// TIA Portal project "HW_2000528_main_V18" (V18)

(* hardware
DEVICE "GSD device_4"  GSD.Device.PN
   slot 0: "Rack"  Rack  V1.0
   slot 0: "CPX_WP5_L"  CPX Rev 30  TN 197330  V4.2.30
      slot 0: "CPX Rev 30"  CPX Rev 30
      slot 1: "PN-IO Interface"  PN-IO Interface
         slot 1: "Port 1"  Port 1
         slot 2: "Port 2"  Port 2
   slot 1: "FB33 PNIO Module_1"  FB33 PNIO Module  TN 548755, CPX-FB33, Code F33
      slot 0: "FB33 PNIO Module"  FB33 PNIO Module
   slot 2: "MPA1S VMPA1-FB-EMS-8 [8DO]_1"  MPA1S VMPA1-FB-EMS-8 [8DO]  TN 533360, VMPA1-FB-EMS-8, Code A
      slot 0: "MPA1S VMPA1-FB-EMS-8 [8DO]"  MPA1S VMPA1-FB-EMS-8 [8DO]
   slot 3: "MPA1S VMPA1-FB-EMS-8 [8DO]_2"  MPA1S VMPA1-FB-EMS-8 [8DO]  TN 533360, VMPA1-FB-EMS-8, Code A
      slot 0: "MPA1S VMPA1-FB-EMS-8 [8DO]"  MPA1S VMPA1-FB-EMS-8 [8DO]
   slot 4: "MPA1S VMPA1-FB-EMS-8 [8DO]_3"  MPA1S VMPA1-FB-EMS-8 [8DO]  TN 533360, VMPA1-FB-EMS-8, Code A
      slot 0: "MPA1S VMPA1-FB-EMS-8 [8DO]"  MPA1S VMPA1-FB-EMS-8 [8DO]
DEVICE "GSD device_2"  GSD.Device.PN
   slot 0: "WP002-DM260-L"  DataMan 260  DMR-260#-#0  5.5.0
      slot 0: "DataMan 260"  DataMan 260
      slot 1: "Interface"  Interface
         slot 1: "Port 1"  Port 1
   slot 0: "Rack"  Rack  V1.0
   slot 1: "Acquisition Control_1"  Acquisition Control
      slot 0: "Acquisition Control"  Acquisition Control
   slot 2: "Acquisition Status_1"  Acquisition Status
      slot 0: "Acquisition Status"  Acquisition Status
   slot 3: "Results Control_1"  Results Control
      slot 0: "Results Control"  Results Control
   slot 4: "Results Status_1"  Results Status
      slot 0: "Results Status"  Results Status
   slot 5: "Soft Event Control_1"  Soft Event Control
      slot 0: "Soft Event Control"  Soft Event Control
   slot 6: "User Data - 64 bytes_1"  User Data - 64 bytes
      slot 0: "User Data - 64 bytes"  User Data - 64 bytes
   slot 7: "Result Data - 64 bytes_1"  Result Data - 64 bytes
      slot 0: "Result Data - 64 bytes"  Result Data - 64 bytes
DEVICE "ET 200SP station_5"  ET 200SP-Station
   slot 0: "R6_L"  IM 155-6 PN ST  6ES7 155-6AU01-0BN0  V4.1
   slot 0: "Rack_0"  Rack  6ES5 710-8MAx1
   slot 1: "DI 16x24VDC ST_1"  DI 16x24VDC ST  6ES7 131-6BH01-0BA0  V0.0
      slot 1: "DI 16x24VDC ST_1"  DI 16x24VDC ST
   slot 2: "DI 16x24VDC ST_2"  DI 16x24VDC ST  6ES7 131-6BH01-0BA0  V0.0
      slot 1: "DI 16x24VDC ST_2"  DI 16x24VDC ST
   slot 3: "DQ 16x24VDC/0.5A ST_1"  DQ 16x24VDC/0.5A ST  6ES7 132-6BH01-0BA0  V0.0
      slot 1: "DQ 16x24VDC/0.5A ST_1"  DQ 16x24VDC/0.5A ST
   slot 4: "DQ 16x24VDC/0.5A ST_2"  DQ 16x24VDC/0.5A ST  6ES7 132-6BH01-0BA0  V0.0
      slot 1: "DQ 16x24VDC/0.5A ST_2"  DQ 16x24VDC/0.5A ST
   slot 5: "Server module_1"  Server module  6ES7 193-6PA00-0AA0  V1.1
      slot 1: "Server module_1"  Server module
   slot 127: "BA 2xRJ45"  BA 2xRJ45  6ES7 193-6AR00-0AA0  V0.0
      slot 1: "Port_1"  X1 P1 R  6ES7 193-6AR00-0AA0  V0.0
      slot 2: "Port_2"  X1 P2 R  6ES7 193-6AR00-0AA0  V0.0
DEVICE "ET 200SP station_4"  ET 200SP-Station
   slot 0: "R2A1_L"  IM 155-6 PN ST  6ES7 155-6AU01-0BN0  V4.1
   slot 0: "Rack_0"  Rack  6ES5 710-8MAx1
   slot 1: "AI 4xU/I 2-wire ST_1"  AI 4xU/I 2-wire ST  6ES7 134-6HD01-0BA1  V2.0
      slot 1: "AI 4xU/I 2-wire ST_1"  AI 4xU/I 2-wire ST
   slot 2: "DI 16x24VDC ST_1"  DI 16x24VDC ST  6ES7 131-6BH01-0BA0  V0.0
      slot 1: "DI 16x24VDC ST_1"  DI 16x24VDC ST
   slot 3: "DI 16x24VDC ST_2"  DI 16x24VDC ST  6ES7 131-6BH01-0BA0  V0.0
      slot 1: "DI 16x24VDC ST_2"  DI 16x24VDC ST
   slot 4: "DI 16x24VDC ST_3"  DI 16x24VDC ST  6ES7 131-6BH01-0BA0  V0.0
      slot 1: "DI 16x24VDC ST_3"  DI 16x24VDC ST
   slot 5: "DI 16x24VDC ST_4"  DI 16x24VDC ST  6ES7 131-6BH01-0BA0  V0.0
      slot 1: "DI 16x24VDC ST_4"  DI 16x24VDC ST
   slot 6: "DI 16x24VDC ST_5"  DI 16x24VDC ST  6ES7 131-6BH01-0BA0  V0.0
      slot 1: "DI 16x24VDC ST_5"  DI 16x24VDC ST
   slot 7: "DI 16x24VDC ST_6"  DI 16x24VDC ST  6ES7 131-6BH01-0BA0  V0.0
      slot 1: "DI 16x24VDC ST_6"  DI 16x24VDC ST
   slot 8: "DQ 16x24VDC/0.5A ST_1"  DQ 16x24VDC/0.5A ST  6ES7 132-6BH01-0BA0  V0.0
      slot 1: "DQ 16x24VDC/0.5A ST_1"  DQ 16x24VDC/0.5A ST
   slot 9: "DQ 16x24VDC/0.5A ST_2"  DQ 16x24VDC/0.5A ST  6ES7 132-6BH01-0BA0  V0.0
      slot 1: "DQ 16x24VDC/0.5A ST_2"  DQ 16x24VDC/0.5A ST
   slot 10: "DQ 16x24VDC/0.5A ST_3"  DQ 16x24VDC/0.5A ST  6ES7 132-6BH01-0BA0  V0.0
      slot 1: "DQ 16x24VDC/0.5A ST_3"  DQ 16x24VDC/0.5A ST
   slot 11: "TM Pulse 2x24V_1"  TM Pulse 2x24V  6ES7 138-6DB00-0BB1  V1.0
      slot 1: "TM Pulse 2x24V_1"  TM Pulse 2x24V
   slot 12: "Server module_1"  Server module  6ES7 193-6PA00-0AA0  V1.1
      slot 1: "Server module_1"  Server module
   slot 127: "BA 2xRJ45"  BA 2xRJ45  6ES7 193-6AR00-0AA0  V0.0
      slot 1: "Port_1"  X1 P1 R  6ES7 193-6AR00-0AA0  V0.0
      slot 2: "Port_2"  X1 P2 R  6ES7 193-6AR00-0AA0  V0.0
DEVICE "ET 200SP station_3"  ET 200SP-Station
   slot 0: "R1A1_L"  IM 155-6 PN ST  6ES7 155-6AU01-0BN0  V4.1
   slot 0: "Rack_0"  Rack  6ES5 710-8MAx1
   slot 1: "DI 16x24VDC ST_1"  DI 16x24VDC ST  6ES7 131-6BH01-0BA0  V0.0
      slot 1: "DI 16x24VDC ST_1"  DI 16x24VDC ST
   slot 2: "DI 16x24VDC ST_2"  DI 16x24VDC ST  6ES7 131-6BH01-0BA0  V0.0
      slot 1: "DI 16x24VDC ST_2"  DI 16x24VDC ST
   slot 3: "DI 16x24VDC ST_3"  DI 16x24VDC ST  6ES7 131-6BH01-0BA0  V0.0
      slot 1: "DI 16x24VDC ST_3"  DI 16x24VDC ST
   slot 4: "DI 16x24VDC ST_4"  DI 16x24VDC ST  6ES7 131-6BH01-0BA0  V0.0
      slot 1: "DI 16x24VDC ST_4"  DI 16x24VDC ST
   slot 5: "DQ 16x24VDC/0.5A ST_1"  DQ 16x24VDC/0.5A ST  6ES7 132-6BH01-0BA0  V0.0
      slot 1: "DQ 16x24VDC/0.5A ST_1"  DQ 16x24VDC/0.5A ST
   slot 6: "DQ 16x24VDC/0.5A ST_2"  DQ 16x24VDC/0.5A ST  6ES7 132-6BH01-0BA0  V0.0
      slot 1: "DQ 16x24VDC/0.5A ST_2"  DQ 16x24VDC/0.5A ST
   slot 7: "DQ 16x24VDC/0.5A ST_3"  DQ 16x24VDC/0.5A ST  6ES7 132-6BH01-0BA0  V0.0
      slot 1: "DQ 16x24VDC/0.5A ST_3"  DQ 16x24VDC/0.5A ST
   slot 8: "Server module_1"  Server module  6ES7 193-6PA00-0AA0  V1.1
      slot 1: "Server module_1"  Server module
   slot 127: "BA 2xRJ45"  BA 2xRJ45  6ES7 193-6AR00-0AA0  V0.0
      slot 1: "Port_1"  X1 P1 R  6ES7 193-6AR00-0AA0  V0.0
      slot 2: "Port_2"  X1 P2 R  6ES7 193-6AR00-0AA0  V0.0
DEVICE "ET 200SP station_2"  ET 200SP-Station
   slot 0: "R0_L"  IM 155-6 PN ST  6ES7 155-6AU01-0BN0  V4.1
   slot 0: "Rack_0"  Rack  6ES5 710-8MAx1
   slot 1: "DI 16x24VDC ST_1"  DI 16x24VDC ST  6ES7 131-6BH01-0BA0  V0.0
      slot 1: "DI 16x24VDC ST_1"  DI 16x24VDC ST
   slot 2: "DI 16x24VDC ST_2"  DI 16x24VDC ST  6ES7 131-6BH01-0BA0  V0.0
      slot 1: "DI 16x24VDC ST_2"  DI 16x24VDC ST
   slot 3: "DI 16x24VDC ST_3"  DI 16x24VDC ST  6ES7 131-6BH01-0BA0  V0.0
      slot 1: "DI 16x24VDC ST_3"  DI 16x24VDC ST
   slot 4: "DI 16x24VDC ST_4"  DI 16x24VDC ST  6ES7 131-6BH01-0BA0  V0.0
      slot 1: "DI 16x24VDC ST_4"  DI 16x24VDC ST
   slot 5: "DI 16x24VDC ST_5"  DI 16x24VDC ST  6ES7 131-6BH01-0BA0  V0.0
      slot 1: "DI 16x24VDC ST_5"  DI 16x24VDC ST
   slot 6: "DI 16x24VDC ST_6"  DI 16x24VDC ST  6ES7 131-6BH01-0BA0  V0.0
      slot 1: "DI 16x24VDC ST_6"  DI 16x24VDC ST
   slot 7: "DQ 16x24VDC/0.5A ST_1"  DQ 16x24VDC/0.5A ST  6ES7 132-6BH01-0BA0  V0.0
      slot 1: "DQ 16x24VDC/0.5A ST_1"  DQ 16x24VDC/0.5A ST
   slot 8: "DQ 16x24VDC/0.5A ST_2"  DQ 16x24VDC/0.5A ST  6ES7 132-6BH01-0BA0  V0.0
      slot 1: "DQ 16x24VDC/0.5A ST_2"  DQ 16x24VDC/0.5A ST
   slot 9: "DQ 16x24VDC/0.5A ST_3"  DQ 16x24VDC/0.5A ST  6ES7 132-6BH01-0BA0  V0.0
      slot 1: "DQ 16x24VDC/0.5A ST_3"  DQ 16x24VDC/0.5A ST
   slot 10: "DQ 16x24VDC/0.5A ST_4"  DQ 16x24VDC/0.5A ST  6ES7 132-6BH01-0BA0  V0.0
      slot 1: "DQ 16x24VDC/0.5A ST_4"  DQ 16x24VDC/0.5A ST
   slot 11: "DQ 16x24VDC/0.5A ST_5"  DQ 16x24VDC/0.5A ST  6ES7 132-6BH01-0BA0  V0.0
      slot 1: "DQ 16x24VDC/0.5A ST_5"  DQ 16x24VDC/0.5A ST
   slot 12: "DI 8x24VDC ST_1"  DI 8x24VDC ST  6ES7 131-6BF01-0BA0  V0.0
      slot 1: "DI 8x24VDC ST_1"  DI 8x24VDC ST
   slot 13: "DI 8x24VDC ST_2"  DI 8x24VDC ST  6ES7 131-6BF01-0BA0  V0.0
      slot 1: "DI 8x24VDC ST_2"  DI 8x24VDC ST
   slot 14: "DI 8x24VDC ST_3"  DI 8x24VDC ST  6ES7 131-6BF01-0BA0  V0.0
      slot 1: "DI 8x24VDC ST_3"  DI 8x24VDC ST
   slot 15: "DI 8x24VDC ST_4"  DI 8x24VDC ST  6ES7 131-6BF01-0BA0  V0.0
      slot 1: "DI 8x24VDC ST_4"  DI 8x24VDC ST
   slot 16: "DI 16x24VDC ST_7"  DI 16x24VDC ST  6ES7 131-6BH01-0BA0  V0.0
      slot 1: "DI 16x24VDC ST_7"  DI 16x24VDC ST
   slot 17: "Server module_1"  Server module  6ES7 193-6PA00-0AA0  V1.1
      slot 1: "Server module_1"  Server module
   slot 127: "BA 2xRJ45"  BA 2xRJ45  6ES7 193-6AR00-0AA0  V0.0
      slot 1: "Port_1"  X1 P1 R  6ES7 193-6AR00-0AA0  V0.0
      slot 2: "Port_2"  X1 P2 R  6ES7 193-6AR00-0AA0  V0.0
DEVICE "ET 200SP station_1"  ET 200SP-Station
   slot 0: "R5A1_L"  IM 155-6 PN ST  6ES7 155-6AU01-0BN0  V4.1
   slot 0: "Rack_0"  Rack  6ES5 710-8MAx1
   slot 1: "CM PtP_1"  CM PtP  6ES7 137-6AA00-0BA0  V1.0
      slot 1: "CM PtP_1"  CM PtP Sub
   slot 2: "AI 4xU/I 2-wire ST_1"  AI 4xU/I 2-wire ST  6ES7 134-6HD01-0BA1  V2.0
      slot 1: "AI 4xU/I 2-wire ST_1"  AI 4xU/I 2-wire ST
   slot 3: "AI 4xU/I 2-wire ST_2"  AI 4xU/I 2-wire ST  6ES7 134-6HD01-0BA1  V2.0
      slot 1: "AI 4xU/I 2-wire ST_2"  AI 4xU/I 2-wire ST
   slot 4: "AQ 4xU/I ST_1"  AQ 4xU/I ST  6ES7 135-6HD00-0BA1  V1.1
      slot 1: "AQ 4xU/I ST_1"  AQ 4xU/I ST
   slot 5: "DI 16x24VDC ST_1"  DI 16x24VDC ST  6ES7 131-6BH01-0BA0  V0.0
      slot 1: "DI 16x24VDC ST_1"  DI 16x24VDC ST
   slot 6: "DI 16x24VDC ST_2"  DI 16x24VDC ST  6ES7 131-6BH01-0BA0  V0.0
      slot 1: "DI 16x24VDC ST_2"  DI 16x24VDC ST
   slot 7: "DI 16x24VDC ST_3"  DI 16x24VDC ST  6ES7 131-6BH01-0BA0  V0.0
      slot 1: "DI 16x24VDC ST_3"  DI 16x24VDC ST
   slot 8: "DI 16x24VDC ST_4"  DI 16x24VDC ST  6ES7 131-6BH01-0BA0  V0.0
      slot 1: "DI 16x24VDC ST_4"  DI 16x24VDC ST
   slot 9: "DI 16x24VDC ST_5"  DI 16x24VDC ST  6ES7 131-6BH01-0BA0  V0.0
      slot 1: "DI 16x24VDC ST_5"  DI 16x24VDC ST
   slot 10: "DQ 16x24VDC/0.5A ST_1"  DQ 16x24VDC/0.5A ST  6ES7 132-6BH01-0BA0  V0.0
      slot 1: "DQ 16x24VDC/0.5A ST_1"  DQ 16x24VDC/0.5A ST
   slot 11: "DQ 16x24VDC/0.5A ST_2"  DQ 16x24VDC/0.5A ST  6ES7 132-6BH01-0BA0  V0.0
      slot 1: "DQ 16x24VDC/0.5A ST_2"  DQ 16x24VDC/0.5A ST
   slot 12: "DQ 16x24VDC/0.5A ST_3"  DQ 16x24VDC/0.5A ST  6ES7 132-6BH01-0BA0  V0.0
      slot 1: "DQ 16x24VDC/0.5A ST_3"  DQ 16x24VDC/0.5A ST
   slot 13: "DQ 16x24VDC/0.5A ST_4"  DQ 16x24VDC/0.5A ST  6ES7 132-6BH01-0BA0  V0.0
      slot 1: "DQ 16x24VDC/0.5A ST_4"  DQ 16x24VDC/0.5A ST
   slot 14: "TM Pulse 2x24V_1"  TM Pulse 2x24V  6ES7 138-6DB00-0BB1  V1.0
      slot 1: "TM Pulse 2x24V_1"  TM Pulse 2x24V
   slot 15: "TM Pulse 2x24V_2"  TM Pulse 2x24V  6ES7 138-6DB00-0BB1  V1.0
      slot 1: "TM Pulse 2x24V_2"  TM Pulse 2x24V
   slot 16: "Server module_1"  Server module  6ES7 193-6PA00-0AA0  V1.1
      slot 1: "Server module_1"  Server module
   slot 127: "BA 2xRJ45"  BA 2xRJ45  6ES7 193-6AR00-0AA0  V0.0
      slot 1: "Port_1"  X1 P1 R  6ES7 193-6AR00-0AA0  V0.0
      slot 2: "Port_2"  X1 P2 R  6ES7 193-6AR00-0AA0  V0.0
DEVICE "GSD device_5"  GSD.Device.PN
   slot 0: "WP001-DM260-L"  DataMan 260  DMR-260#-#0  5.5.0
      slot 0: "DataMan 260"  DataMan 260
      slot 1: "Interface"  Interface
         slot 1: "Port 1"  Port 1
   slot 0: "Rack"  Rack  V1.0
   slot 1: "Acquisition Control_1"  Acquisition Control
      slot 0: "Acquisition Control"  Acquisition Control
   slot 2: "Acquisition Status_1"  Acquisition Status
      slot 0: "Acquisition Status"  Acquisition Status
   slot 3: "Results Control_1"  Results Control
      slot 0: "Results Control"  Results Control
   slot 4: "Results Status_1"  Results Status
      slot 0: "Results Status"  Results Status
   slot 5: "Soft Event Control_1"  Soft Event Control
      slot 0: "Soft Event Control"  Soft Event Control
   slot 6: "User Data - 64 bytes_1"  User Data - 64 bytes
      slot 0: "User Data - 64 bytes"  User Data - 64 bytes
   slot 7: "Result Data - 64 bytes_1"  Result Data - 64 bytes
      slot 0: "Result Data - 64 bytes"  Result Data - 64 bytes
DEVICE "GSD device_1"  GSD.Device.PN
   slot 0: "UR5_st4_L"  V1.0  00000
      slot 0: "V1.0"  V1.0
      slot 1: "Interface"  Interface
         slot 1: "RJ45 10/100 MBit/s"  RJ45 10/100 MBit/s
   slot 0: "Rack"  Rack  V1.0
   slot 1: "1_T2O State"  1_T2O State  1.0
      slot 0: "1_T2O State"  1_T2O State
   slot 2: "2_T2O IO"  2_T2O IO  1.0
      slot 0: "2_T2O IO"  2_T2O IO
   slot 3: "3_T2O Joints"  3_T2O Joints  1.0
      slot 0: "3_T2O Joints"  3_T2O Joints
   slot 4: "4_T2O TCP"  4_T2O TCP  1.0
      slot 0: "4_T2O TCP"  4_T2O TCP
   slot 5: "5_T2O General Purpose Bit Registers"  5_T2O General Purpose Bit Registers  1.0
      slot 0: "5_T2O General Purpose Bit Registers"  5_T2O General Purpose Bit Registers
   slot 6: "6_T2O General Purpose Int Registers"  6_T2O General Purpose Int Registers  1.0
      slot 0: "6_T2O General Purpose Int Registers"  6_T2O General Purpose Int Registers
   slot 7: "7_T2O General Purpose Float Registers"  7_T2O General Purpose Float Registers  1.0
      slot 0: "7_T2O General Purpose Float Registers"  7_T2O General Purpose Float Registers
   slot 8: "8_O2T Robot IO"  8_O2T Robot IO  1.0
      slot 0: "8_O2T Robot IO"  8_O2T Robot IO
   slot 9: "9_O2T General Purpose Registers 1"  9_O2T General Purpose Registers 1  1.0
      slot 0: "9_O2T General Purpose Registers 1"  9_O2T General Purpose Registers 1
   slot 10: "10_O2T General Purpose Registers 2"  10_O2T General Purpose Registers 2  1.0
      slot 0: "10_O2T General Purpose Registers 2"  10_O2T General Purpose Registers 2
DEVICE "GSD device_6"  GSD.Device.PN
   slot 0: "Rack"  Rack  V1.0
   slot 0: "CPX_TS_L"  CPX Rev 30  TN 197330  V4.2.30
      slot 0: "CPX Rev 30"  CPX Rev 30
      slot 1: "PN-IO Interface"  PN-IO Interface
         slot 1: "Port 1"  Port 1
         slot 2: "Port 2"  Port 2
   slot 1: "FB33 PNIO Module_1"  FB33 PNIO Module  TN 548755, CPX-FB33, Code F33
      slot 0: "FB33 PNIO Module"  FB33 PNIO Module
   slot 2: "MPA2S VMPA2-FB-EMS-4 [4DO]_1"  MPA2S VMPA2-FB-EMS-4 [4DO]  TN 537983, VMPA2-FB-EMS-4, Code B
      slot 0: "MPA2S VMPA2-FB-EMS-4 [4DO]"  MPA2S VMPA2-FB-EMS-4 [4DO]
   slot 3: "MPA2G VMPA2-FB-EMG-4 [4DO]_1"  MPA2G VMPA2-FB-EMG-4 [4DO]  TN 537984, VMPA2-FB-EMG-4, Code BH
      slot 0: "MPA2G VMPA2-FB-EMG-4 [4DO]"  MPA2G VMPA2-FB-EMG-4 [4DO]
   slot 4: "MPA1G VMPA1-FB-EMG-8 [8DO]_2"  MPA1G VMPA1-FB-EMG-8 [8DO]  TN 533361, VMPA1-FB-EMG-8, Code AH
      slot 0: "MPA1G VMPA1-FB-EMG-8 [8DO]"  MPA1G VMPA1-FB-EMG-8 [8DO]
   slot 5: "MPA1G VMPA1-FB-EMG-8 [8DO]_3"  MPA1G VMPA1-FB-EMG-8 [8DO]  TN 533361, VMPA1-FB-EMG-8, Code AH
      slot 0: "MPA1G VMPA1-FB-EMG-8 [8DO]"  MPA1G VMPA1-FB-EMG-8 [8DO]
   slot 6: "MPA1G VMPA1-FB-EMG-8 [8DO]_4"  MPA1G VMPA1-FB-EMG-8 [8DO]  TN 533361, VMPA1-FB-EMG-8, Code AH
      slot 0: "MPA1G VMPA1-FB-EMG-8 [8DO]"  MPA1G VMPA1-FB-EMG-8 [8DO]
   slot 7: "MPA1G VMPA1-FB-EMG-8 [8DO]_5"  MPA1G VMPA1-FB-EMG-8 [8DO]  TN 533361, VMPA1-FB-EMG-8, Code AH
      slot 0: "MPA1G VMPA1-FB-EMG-8 [8DO]"  MPA1G VMPA1-FB-EMG-8 [8DO]
   slot 8: "MPA1G VMPA1-FB-EMG-8 [8DO]_6"  MPA1G VMPA1-FB-EMG-8 [8DO]  TN 533361, VMPA1-FB-EMG-8, Code AH
      slot 0: "MPA1G VMPA1-FB-EMG-8 [8DO]"  MPA1G VMPA1-FB-EMG-8 [8DO]
DEVICE "GSD device_7"  GSD.Device.PN
   slot 0: "Rack"  Rack  V1.0
   slot 0: "CPX_WP2_L"  CPX Rev 30  TN 197330  V4.2.30
      slot 0: "CPX Rev 30"  CPX Rev 30
      slot 1: "PN-IO Interface"  PN-IO Interface
         slot 1: "Port 1"  Port 1
         slot 2: "Port 2"  Port 2
   slot 1: "FB33 PNIO Module_1"  FB33 PNIO Module  TN 548755, CPX-FB33, Code F33
      slot 0: "FB33 PNIO Module"  FB33 PNIO Module
   slot 2: "MPA1S VMPA1-FB-EMS-8 [8DO]_1"  MPA1S VMPA1-FB-EMS-8 [8DO]  TN 533360, VMPA1-FB-EMS-8, Code A
      slot 0: "MPA1S VMPA1-FB-EMS-8 [8DO]"  MPA1S VMPA1-FB-EMS-8 [8DO]
   slot 3: "MPA1S VMPA1-FB-EMS-8 [8DO]_2"  MPA1S VMPA1-FB-EMS-8 [8DO]  TN 533360, VMPA1-FB-EMS-8, Code A
      slot 0: "MPA1S VMPA1-FB-EMS-8 [8DO]"  MPA1S VMPA1-FB-EMS-8 [8DO]
   slot 4: "MPA1S VMPA1-FB-EMS-8 [8DO]_3"  MPA1S VMPA1-FB-EMS-8 [8DO]  TN 533360, VMPA1-FB-EMS-8, Code A
      slot 0: "MPA1S VMPA1-FB-EMS-8 [8DO]"  MPA1S VMPA1-FB-EMS-8 [8DO]
   slot 5: "MPA1G VMPA1-FB-EMG-8 [8DO]_3"  MPA1G VMPA1-FB-EMG-8 [8DO]  TN 533361, VMPA1-FB-EMG-8, Code AH
      slot 0: "MPA1G VMPA1-FB-EMG-8 [8DO]"  MPA1G VMPA1-FB-EMG-8 [8DO]
DEVICE "GSD device_9"  GSD.Device.PN
   slot 0: "Rack"  Rack  V1.0
   slot 0: "fx0-gpnt_L"  FX0-GPNT V2  1044074  V2.12.00
      slot 0: "FX0-GPNT V2_1"  FX0-GPNT V2
      slot 1: "FX0-GPNT V2"  FX0-GPNT V2
         slot 1: "Port 1"  Port 1
         slot 2: "Port 2"  Port 2
   slot 1: "Input Data Block 1_1"  Input Data Block 1
      slot 0: "Input Data Block 1"  Input Data Block 1
   slot 2: "Input Data Block 2_1"  Input Data Block 2
      slot 0: "Input Data Block 2"  Input Data Block 2
   slot 3: "Input Data Block 3_1"  Input Data Block 3
      slot 0: "Input Data Block 3"  Input Data Block 3
   slot 4: "Input Data Block 4_1"  Input Data Block 4
      slot 0: "Input Data Block 4"  Input Data Block 4
   slot 5: "Input Data Block 5_1"  Input Data Block 5
      slot 0: "Input Data Block 5"  Input Data Block 5
   slot 6: "Output Data Block 1_1"  Output Data Block 1
      slot 0: "Output Data Block 1"  Output Data Block 1
   slot 7: "Output Data Block 2_1"  Output Data Block 2
      slot 0: "Output Data Block 2"  Output Data Block 2
   slot 8: "Output Data Block 3_1"  Output Data Block 3
      slot 0: "Output Data Block 3"  Output Data Block 3
   slot 9: "Output Data Block 4_1"  Output Data Block 4
      slot 0: "Output Data Block 4"  Output Data Block 4
   slot 10: "Output Data Block 5_1"  Output Data Block 5
      slot 0: "Output Data Block 5"  Output Data Block 5
DEVICE "GSD device_8"  GSD.Device.PN
   slot 0: "Rack"  Rack  V1.0
   slot 0: "WP004-DM260-L"  DataMan 260  DMR-260#-#0  5.5.0
      slot 0: "DataMan 260"  DataMan 260
      slot 1: "Interface"  Interface
         slot 1: "Port 1"  Port 1
   slot 1: "Acquisition Control_1"  Acquisition Control
      slot 0: "Acquisition Control"  Acquisition Control
   slot 2: "Acquisition Status_1"  Acquisition Status
      slot 0: "Acquisition Status"  Acquisition Status
   slot 3: "Results Control_1"  Results Control
      slot 0: "Results Control"  Results Control
   slot 4: "Results Status_1"  Results Status
      slot 0: "Results Status"  Results Status
   slot 5: "Soft Event Control_1"  Soft Event Control
      slot 0: "Soft Event Control"  Soft Event Control
   slot 6: "User Data - 64 bytes_1"  User Data - 64 bytes
      slot 0: "User Data - 64 bytes"  User Data - 64 bytes
   slot 7: "Result Data - 64 bytes_1"  Result Data - 64 bytes
      slot 0: "Result Data - 64 bytes"  Result Data - 64 bytes
DEVICE "GSD device_10"  GSD.Device.PN
   slot 0: "Rack"  Rack  V1.0
   slot 0: "WP0031-DM260-L"  DataMan 260  DMR-260#-#0  5.5.0
      slot 0: "DataMan 260"  DataMan 260
      slot 1: "Interface"  Interface
         slot 1: "Port 1"  Port 1
   slot 1: "Acquisition Control_1"  Acquisition Control
      slot 0: "Acquisition Control"  Acquisition Control
   slot 2: "Acquisition Status_1"  Acquisition Status
      slot 0: "Acquisition Status"  Acquisition Status
   slot 3: "Results Control_1"  Results Control
      slot 0: "Results Control"  Results Control
   slot 4: "Results Status_1"  Results Status
      slot 0: "Results Status"  Results Status
   slot 5: "Soft Event Control_1"  Soft Event Control
      slot 0: "Soft Event Control"  Soft Event Control
   slot 6: "User Data - 64 bytes_1"  User Data - 64 bytes
      slot 0: "User Data - 64 bytes"  User Data - 64 bytes
   slot 7: "Result Data - 64 bytes_1"  Result Data - 64 bytes
      slot 0: "Result Data - 64 bytes"  Result Data - 64 bytes
DEVICE "GSD device_11"  GSD.Device.PN
   slot 0: "Rack"  Rack  V1.0
   slot 0: "WP003-DM260-L"  DataMan 260  DMR-260#-#0  5.5.0
      slot 0: "DataMan 260"  DataMan 260
      slot 1: "Interface"  Interface
         slot 1: "Port 1"  Port 1
   slot 1: "Acquisition Control_1"  Acquisition Control
      slot 0: "Acquisition Control"  Acquisition Control
   slot 2: "Acquisition Status_1"  Acquisition Status
      slot 0: "Acquisition Status"  Acquisition Status
   slot 3: "Results Control_1"  Results Control
      slot 0: "Results Control"  Results Control
   slot 4: "Results Status_1"  Results Status
      slot 0: "Results Status"  Results Status
   slot 5: "Soft Event Control_1"  Soft Event Control
      slot 0: "Soft Event Control"  Soft Event Control
   slot 6: "User Data - 64 bytes_1"  User Data - 64 bytes
      slot 0: "User Data - 64 bytes"  User Data - 64 bytes
   slot 7: "Result Data - 64 bytes_1"  Result Data - 64 bytes
      slot 0: "Result Data - 64 bytes"  Result Data - 64 bytes
DEVICE "GSD device_12"  GSD.Device.PN
   slot 0: "Rack"  Rack  V1.0
   slot 0: "WP005-DM260-L"  DataMan 260  DMR-260#-#0  5.5.0
      slot 0: "DataMan 260"  DataMan 260
      slot 1: "Interface"  Interface
         slot 1: "Port 1"  Port 1
   slot 1: "Acquisition Control_1"  Acquisition Control
      slot 0: "Acquisition Control"  Acquisition Control
   slot 2: "Acquisition Status_1"  Acquisition Status
      slot 0: "Acquisition Status"  Acquisition Status
   slot 3: "Results Control_1"  Results Control
      slot 0: "Results Control"  Results Control
   slot 4: "Results Status_1"  Results Status
      slot 0: "Results Status"  Results Status
   slot 5: "Soft Event Control_1"  Soft Event Control
      slot 0: "Soft Event Control"  Soft Event Control
   slot 6: "User Data - 64 bytes_1"  User Data - 64 bytes
      slot 0: "User Data - 64 bytes"  User Data - 64 bytes
   slot 7: "Result Data - 64 bytes_1"  Result Data - 64 bytes
      slot 0: "Result Data - 64 bytes"  Result Data - 64 bytes
DEVICE "GSD device_13"  GSD.Device.PN
   slot 0: "Rack"  Rack  V1.0
   slot 0: "WP006-DM260-L"  DataMan 260  DMR-260#-#0  5.5.0
      slot 0: "DataMan 260"  DataMan 260
      slot 1: "Interface"  Interface
         slot 1: "Port 1"  Port 1
   slot 1: "Acquisition Control_1"  Acquisition Control
      slot 0: "Acquisition Control"  Acquisition Control
   slot 2: "Acquisition Status_1"  Acquisition Status
      slot 0: "Acquisition Status"  Acquisition Status
   slot 3: "Results Control_1"  Results Control
      slot 0: "Results Control"  Results Control
   slot 4: "Results Status_1"  Results Status
      slot 0: "Results Status"  Results Status
   slot 5: "Soft Event Control_1"  Soft Event Control
      slot 0: "Soft Event Control"  Soft Event Control
   slot 6: "User Data - 64 bytes_1"  User Data - 64 bytes
      slot 0: "User Data - 64 bytes"  User Data - 64 bytes
   slot 7: "Result Data - 64 bytes_1"  Result Data - 64 bytes
      slot 0: "Result Data - 64 bytes"  Result Data - 64 bytes
DEVICE "GSD device_16"  GSD.Device.PN
   slot 0: "Rack"  Rack  V1.0
   slot 0: "WP001-DM8050-L"  DataMan 8000  DMR-8#00-0#00  5.4.2
      slot 0: "DataMan 8000"  DataMan 8000
      slot 1: "Interface"  Interface
         slot 1: "Port 1"  Port 1
   slot 1: "Acquisition Control_1"  Acquisition Control
      slot 0: "Acquisition Control"  Acquisition Control
   slot 2: "Acquisition Status_1"  Acquisition Status
      slot 0: "Acquisition Status"  Acquisition Status
   slot 3: "Results Control_1"  Results Control
      slot 0: "Results Control"  Results Control
   slot 4: "Results Status_1"  Results Status
      slot 0: "Results Status"  Results Status
   slot 5: "Soft Event Control_1"  Soft Event Control
      slot 0: "Soft Event Control"  Soft Event Control
   slot 6: "User Data - 64 bytes_1"  User Data - 64 bytes
      slot 0: "User Data - 64 bytes"  User Data - 64 bytes
   slot 7: "Result Data - 64 bytes_1"  Result Data - 64 bytes
      slot 0: "Result Data - 64 bytes"  Result Data - 64 bytes
DEVICE "GSD device_17"  GSD.Device.PN
   slot 0: "Rack"  Rack  V1.0
   slot 0: "WP004-DM8050-L"  DataMan 8000  DMR-8#00-0#00  5.4.2
      slot 0: "DataMan 8000"  DataMan 8000
      slot 1: "Interface"  Interface
         slot 1: "Port 1"  Port 1
   slot 1: "Acquisition Control_1"  Acquisition Control
      slot 0: "Acquisition Control"  Acquisition Control
   slot 2: "Acquisition Status_1"  Acquisition Status
      slot 0: "Acquisition Status"  Acquisition Status
   slot 3: "Results Control_1"  Results Control
      slot 0: "Results Control"  Results Control
   slot 4: "Results Status_1"  Results Status
      slot 0: "Results Status"  Results Status
   slot 5: "Soft Event Control_1"  Soft Event Control
      slot 0: "Soft Event Control"  Soft Event Control
   slot 6: "User Data - 64 bytes_1"  User Data - 64 bytes
      slot 0: "User Data - 64 bytes"  User Data - 64 bytes
   slot 7: "Result Data - 64 bytes_1"  Result Data - 64 bytes
      slot 0: "Result Data - 64 bytes"  Result Data - 64 bytes
DEVICE "GSD device_18"  GSD.Device.PN
   slot 0: "Rack"  Rack  V1.0
   slot 0: "fx0-gpnt_R"  FX0-GPNT V2  1044074  V2.12.00
      slot 0: "FX0-GPNT V2_1"  FX0-GPNT V2
      slot 1: "FX0-GPNT V2"  FX0-GPNT V2
         slot 1: "Port 1"  Port 1
         slot 2: "Port 2"  Port 2
   slot 1: "Input Data Block 1_1"  Input Data Block 1
      slot 0: "Input Data Block 1"  Input Data Block 1
   slot 2: "Input Data Block 2_1"  Input Data Block 2
      slot 0: "Input Data Block 2"  Input Data Block 2
   slot 3: "Input Data Block 3_1"  Input Data Block 3
      slot 0: "Input Data Block 3"  Input Data Block 3
   slot 4: "Input Data Block 4_1"  Input Data Block 4
      slot 0: "Input Data Block 4"  Input Data Block 4
   slot 5: "Input Data Block 5_1"  Input Data Block 5
      slot 0: "Input Data Block 5"  Input Data Block 5
   slot 6: "Output Data Block 1_1"  Output Data Block 1
      slot 0: "Output Data Block 1"  Output Data Block 1
   slot 7: "Output Data Block 2_1"  Output Data Block 2
      slot 0: "Output Data Block 2"  Output Data Block 2
   slot 8: "Output Data Block 3_1"  Output Data Block 3
      slot 0: "Output Data Block 3"  Output Data Block 3
   slot 9: "Output Data Block 4_1"  Output Data Block 4
      slot 0: "Output Data Block 4"  Output Data Block 4
   slot 10: "Output Data Block 5_1"  Output Data Block 5
      slot 0: "Output Data Block 5"  Output Data Block 5
DEVICE "ET 200SP station_6"  ET 200SP-Station
   slot 0: "Rack_0"  Rack  6ES5 710-8MAx1
   slot 0: "R0_R"  IM 155-6 PN ST  6ES7 155-6AU01-0BN0  V4.1
   slot 1: "DI 16x24VDC ST_1"  DI 16x24VDC ST  6ES7 131-6BH01-0BA0  V0.0
      slot 1: "DI 16x24VDC ST_1"  DI 16x24VDC ST
   slot 2: "DI 16x24VDC ST_2"  DI 16x24VDC ST  6ES7 131-6BH01-0BA0  V0.0
      slot 1: "DI 16x24VDC ST_2"  DI 16x24VDC ST
   slot 3: "DI 16x24VDC ST_3"  DI 16x24VDC ST  6ES7 131-6BH01-0BA0  V0.0
      slot 1: "DI 16x24VDC ST_3"  DI 16x24VDC ST
   slot 4: "DI 16x24VDC ST_4"  DI 16x24VDC ST  6ES7 131-6BH01-0BA0  V0.0
      slot 1: "DI 16x24VDC ST_4"  DI 16x24VDC ST
   slot 5: "DI 16x24VDC ST_5"  DI 16x24VDC ST  6ES7 131-6BH01-0BA0  V0.0
      slot 1: "DI 16x24VDC ST_5"  DI 16x24VDC ST
   slot 6: "DI 16x24VDC ST_6"  DI 16x24VDC ST  6ES7 131-6BH01-0BA0  V0.0
      slot 1: "DI 16x24VDC ST_6"  DI 16x24VDC ST
   slot 7: "DQ 16x24VDC/0.5A ST_1"  DQ 16x24VDC/0.5A ST  6ES7 132-6BH01-0BA0  V0.0
      slot 1: "DQ 16x24VDC/0.5A ST_1"  DQ 16x24VDC/0.5A ST
   slot 8: "DQ 16x24VDC/0.5A ST_2"  DQ 16x24VDC/0.5A ST  6ES7 132-6BH01-0BA0  V0.0
      slot 1: "DQ 16x24VDC/0.5A ST_2"  DQ 16x24VDC/0.5A ST
   slot 9: "DQ 16x24VDC/0.5A ST_3"  DQ 16x24VDC/0.5A ST  6ES7 132-6BH01-0BA0  V0.0
      slot 1: "DQ 16x24VDC/0.5A ST_3"  DQ 16x24VDC/0.5A ST
   slot 10: "DQ 16x24VDC/0.5A ST_4"  DQ 16x24VDC/0.5A ST  6ES7 132-6BH01-0BA0  V0.0
      slot 1: "DQ 16x24VDC/0.5A ST_4"  DQ 16x24VDC/0.5A ST
   slot 11: "DQ 16x24VDC/0.5A ST_5"  DQ 16x24VDC/0.5A ST  6ES7 132-6BH01-0BA0  V0.0
      slot 1: "DQ 16x24VDC/0.5A ST_5"  DQ 16x24VDC/0.5A ST
   slot 12: "DI 8x24VDC ST_1"  DI 8x24VDC ST  6ES7 131-6BF01-0BA0  V0.0
      slot 1: "DI 8x24VDC ST_1"  DI 8x24VDC ST
   slot 13: "DI 8x24VDC ST_2"  DI 8x24VDC ST  6ES7 131-6BF01-0BA0  V0.0
      slot 1: "DI 8x24VDC ST_2"  DI 8x24VDC ST
   slot 14: "DI 8x24VDC ST_3"  DI 8x24VDC ST  6ES7 131-6BF01-0BA0  V0.0
      slot 1: "DI 8x24VDC ST_3"  DI 8x24VDC ST
   slot 15: "DI 8x24VDC ST_4"  DI 8x24VDC ST  6ES7 131-6BF01-0BA0  V0.0
      slot 1: "DI 8x24VDC ST_4"  DI 8x24VDC ST
   slot 16: "DI 16x24VDC ST_7"  DI 16x24VDC ST  6ES7 131-6BH01-0BA0  V0.0
      slot 1: "DI 16x24VDC ST_7"  DI 16x24VDC ST
   slot 17: "Server module_1"  Server module  6ES7 193-6PA00-0AA0  V1.1
      slot 1: "Server module_1"  Server module
   slot 127: "BA 2xRJ45"  BA 2xRJ45  6ES7 193-6AR00-0AA0  V0.0
      slot 1: "Port_1"  X1 P1 R  6ES7 193-6AR00-0AA0  V0.0
      slot 2: "Port_2"  X1 P2 R  6ES7 193-6AR00-0AA0  V0.0
DEVICE "ET 200SP station_7"  ET 200SP-Station
   slot 0: "Rack_0"  Rack  6ES5 710-8MAx1
   slot 0: "R5A1_R"  IM 155-6 PN ST  6ES7 155-6AU01-0BN0  V4.1
   slot 1: "CM PtP_1"  CM PtP  6ES7 137-6AA00-0BA0  V1.0
      slot 1: "CM PtP_1"  CM PtP Sub
   slot 2: "AI 4xU/I 2-wire ST_1"  AI 4xU/I 2-wire ST  6ES7 134-6HD01-0BA1  V2.0
      slot 1: "AI 4xU/I 2-wire ST_1"  AI 4xU/I 2-wire ST
   slot 3: "AI 4xU/I 2-wire ST_2"  AI 4xU/I 2-wire ST  6ES7 134-6HD01-0BA1  V2.0
      slot 1: "AI 4xU/I 2-wire ST_2"  AI 4xU/I 2-wire ST
   slot 4: "AQ 4xU/I ST_1"  AQ 4xU/I ST  6ES7 135-6HD00-0BA1  V1.1
      slot 1: "AQ 4xU/I ST_1"  AQ 4xU/I ST
   slot 5: "DI 16x24VDC ST_1"  DI 16x24VDC ST  6ES7 131-6BH01-0BA0  V0.0
      slot 1: "DI 16x24VDC ST_1"  DI 16x24VDC ST
   slot 6: "DI 16x24VDC ST_2"  DI 16x24VDC ST  6ES7 131-6BH01-0BA0  V0.0
      slot 1: "DI 16x24VDC ST_2"  DI 16x24VDC ST
   slot 7: "DI 16x24VDC ST_3"  DI 16x24VDC ST  6ES7 131-6BH01-0BA0  V0.0
      slot 1: "DI 16x24VDC ST_3"  DI 16x24VDC ST
   slot 8: "DI 16x24VDC ST_4"  DI 16x24VDC ST  6ES7 131-6BH01-0BA0  V0.0
      slot 1: "DI 16x24VDC ST_4"  DI 16x24VDC ST
   slot 9: "DI 16x24VDC ST_5"  DI 16x24VDC ST  6ES7 131-6BH01-0BA0  V0.0
      slot 1: "DI 16x24VDC ST_5"  DI 16x24VDC ST
   slot 10: "DQ 16x24VDC/0.5A ST_1"  DQ 16x24VDC/0.5A ST  6ES7 132-6BH01-0BA0  V0.0
      slot 1: "DQ 16x24VDC/0.5A ST_1"  DQ 16x24VDC/0.5A ST
   slot 11: "DQ 16x24VDC/0.5A ST_2"  DQ 16x24VDC/0.5A ST  6ES7 132-6BH01-0BA0  V0.0
      slot 1: "DQ 16x24VDC/0.5A ST_2"  DQ 16x24VDC/0.5A ST
   slot 12: "DQ 16x24VDC/0.5A ST_3"  DQ 16x24VDC/0.5A ST  6ES7 132-6BH01-0BA0  V0.0
      slot 1: "DQ 16x24VDC/0.5A ST_3"  DQ 16x24VDC/0.5A ST
   slot 13: "DQ 16x24VDC/0.5A ST_4"  DQ 16x24VDC/0.5A ST  6ES7 132-6BH01-0BA0  V0.0
      slot 1: "DQ 16x24VDC/0.5A ST_4"  DQ 16x24VDC/0.5A ST
   slot 14: "TM Pulse 2x24V_1"  TM Pulse 2x24V  6ES7 138-6DB00-0BB1  V1.0
      slot 1: "TM Pulse 2x24V_1"  TM Pulse 2x24V
   slot 15: "TM Pulse 2x24V_2"  TM Pulse 2x24V  6ES7 138-6DB00-0BB1  V1.0
      slot 1: "TM Pulse 2x24V_2"  TM Pulse 2x24V
   slot 16: "Server module_1"  Server module  6ES7 193-6PA00-0AA0  V1.1
      slot 1: "Server module_1"  Server module
   slot 127: "BA 2xRJ45"  BA 2xRJ45  6ES7 193-6AR00-0AA0  V0.0
      slot 1: "Port_1"  X1 P1 R  6ES7 193-6AR00-0AA0  V0.0
      slot 2: "Port_2"  X1 P2 R  6ES7 193-6AR00-0AA0  V0.0
DEVICE "ET 200SP station_8"  ET 200SP-Station
   slot 0: "Rack_0"  Rack  6ES5 710-8MAx1
   slot 0: "R1A1_R"  IM 155-6 PN ST  6ES7 155-6AU01-0BN0  V4.1
   slot 1: "DI 16x24VDC ST_1"  DI 16x24VDC ST  6ES7 131-6BH01-0BA0  V0.0
      slot 1: "DI 16x24VDC ST_1"  DI 16x24VDC ST
   slot 2: "DI 16x24VDC ST_2"  DI 16x24VDC ST  6ES7 131-6BH01-0BA0  V0.0
      slot 1: "DI 16x24VDC ST_2"  DI 16x24VDC ST
   slot 3: "DI 16x24VDC ST_3"  DI 16x24VDC ST  6ES7 131-6BH01-0BA0  V0.0
      slot 1: "DI 16x24VDC ST_3"  DI 16x24VDC ST
   slot 4: "DI 16x24VDC ST_4"  DI 16x24VDC ST  6ES7 131-6BH01-0BA0  V0.0
      slot 1: "DI 16x24VDC ST_4"  DI 16x24VDC ST
   slot 5: "DQ 16x24VDC/0.5A ST_1"  DQ 16x24VDC/0.5A ST  6ES7 132-6BH01-0BA0  V0.0
      slot 1: "DQ 16x24VDC/0.5A ST_1"  DQ 16x24VDC/0.5A ST
   slot 6: "DQ 16x24VDC/0.5A ST_2"  DQ 16x24VDC/0.5A ST  6ES7 132-6BH01-0BA0  V0.0
      slot 1: "DQ 16x24VDC/0.5A ST_2"  DQ 16x24VDC/0.5A ST
   slot 7: "DQ 16x24VDC/0.5A ST_3"  DQ 16x24VDC/0.5A ST  6ES7 132-6BH01-0BA0  V0.0
      slot 1: "DQ 16x24VDC/0.5A ST_3"  DQ 16x24VDC/0.5A ST
   slot 8: "Server module_1"  Server module  6ES7 193-6PA00-0AA0  V1.1
      slot 1: "Server module_1"  Server module
   slot 127: "BA 2xRJ45"  BA 2xRJ45  6ES7 193-6AR00-0AA0  V0.0
      slot 1: "Port_1"  X1 P1 R  6ES7 193-6AR00-0AA0  V0.0
      slot 2: "Port_2"  X1 P2 R  6ES7 193-6AR00-0AA0  V0.0
DEVICE "ET 200SP station_9"  ET 200SP-Station
   slot 0: "Rack_0"  Rack  6ES5 710-8MAx1
   slot 0: "R2A1_R"  IM 155-6 PN ST  6ES7 155-6AU01-0BN0  V4.1
   slot 1: "AI 4xU/I 2-wire ST_1"  AI 4xU/I 2-wire ST  6ES7 134-6HD01-0BA1  V2.0
      slot 1: "AI 4xU/I 2-wire ST_1"  AI 4xU/I 2-wire ST
   slot 2: "DI 16x24VDC ST_1"  DI 16x24VDC ST  6ES7 131-6BH01-0BA0  V0.0
      slot 1: "DI 16x24VDC ST_1"  DI 16x24VDC ST
   slot 3: "DI 16x24VDC ST_2"  DI 16x24VDC ST  6ES7 131-6BH01-0BA0  V0.0
      slot 1: "DI 16x24VDC ST_2"  DI 16x24VDC ST
   slot 4: "DI 16x24VDC ST_3"  DI 16x24VDC ST  6ES7 131-6BH01-0BA0  V0.0
      slot 1: "DI 16x24VDC ST_3"  DI 16x24VDC ST
   slot 5: "DI 16x24VDC ST_4"  DI 16x24VDC ST  6ES7 131-6BH01-0BA0  V0.0
      slot 1: "DI 16x24VDC ST_4"  DI 16x24VDC ST
   slot 6: "DI 16x24VDC ST_5"  DI 16x24VDC ST  6ES7 131-6BH01-0BA0  V0.0
      slot 1: "DI 16x24VDC ST_5"  DI 16x24VDC ST
   slot 7: "DI 16x24VDC ST_6"  DI 16x24VDC ST  6ES7 131-6BH01-0BA0  V0.0
      slot 1: "DI 16x24VDC ST_6"  DI 16x24VDC ST
   slot 8: "DQ 16x24VDC/0.5A ST_1"  DQ 16x24VDC/0.5A ST  6ES7 132-6BH01-0BA0  V0.0
      slot 1: "DQ 16x24VDC/0.5A ST_1"  DQ 16x24VDC/0.5A ST
   slot 9: "DQ 16x24VDC/0.5A ST_2"  DQ 16x24VDC/0.5A ST  6ES7 132-6BH01-0BA0  V0.0
      slot 1: "DQ 16x24VDC/0.5A ST_2"  DQ 16x24VDC/0.5A ST
   slot 10: "DQ 16x24VDC/0.5A ST_3"  DQ 16x24VDC/0.5A ST  6ES7 132-6BH01-0BA0  V0.0
      slot 1: "DQ 16x24VDC/0.5A ST_3"  DQ 16x24VDC/0.5A ST
   slot 11: "TM Pulse 2x24V_1"  TM Pulse 2x24V  6ES7 138-6DB00-0BB1  V1.0
      slot 1: "TM Pulse 2x24V_1"  TM Pulse 2x24V
   slot 12: "Server module_1"  Server module  6ES7 193-6PA00-0AA0  V1.1
      slot 1: "Server module_1"  Server module
   slot 127: "BA 2xRJ45"  BA 2xRJ45  6ES7 193-6AR00-0AA0  V0.0
      slot 1: "Port_1"  X1 P1 R  6ES7 193-6AR00-0AA0  V0.0
      slot 2: "Port_2"  X1 P2 R  6ES7 193-6AR00-0AA0  V0.0
DEVICE "ET 200SP station_10"  ET 200SP-Station
   slot 0: "Rack_0"  Rack  6ES5 710-8MAx1
   slot 0: "R6_R"  IM 155-6 PN ST  6ES7 155-6AU01-0BN0  V4.1
   slot 1: "DI 16x24VDC ST_1"  DI 16x24VDC ST  6ES7 131-6BH01-0BA0  V0.0
      slot 1: "DI 16x24VDC ST_1"  DI 16x24VDC ST
   slot 2: "DI 16x24VDC ST_2"  DI 16x24VDC ST  6ES7 131-6BH01-0BA0  V0.0
      slot 1: "DI 16x24VDC ST_2"  DI 16x24VDC ST
   slot 3: "DQ 16x24VDC/0.5A ST_1"  DQ 16x24VDC/0.5A ST  6ES7 132-6BH01-0BA0  V0.0
      slot 1: "DQ 16x24VDC/0.5A ST_1"  DQ 16x24VDC/0.5A ST
   slot 4: "DQ 16x24VDC/0.5A ST_2"  DQ 16x24VDC/0.5A ST  6ES7 132-6BH01-0BA0  V0.0
      slot 1: "DQ 16x24VDC/0.5A ST_2"  DQ 16x24VDC/0.5A ST
   slot 5: "Server module_1"  Server module  6ES7 193-6PA00-0AA0  V1.1
      slot 1: "Server module_1"  Server module
   slot 127: "BA 2xRJ45"  BA 2xRJ45  6ES7 193-6AR00-0AA0  V0.0
      slot 1: "Port_1"  X1 P1 R  6ES7 193-6AR00-0AA0  V0.0
      slot 2: "Port_2"  X1 P2 R  6ES7 193-6AR00-0AA0  V0.0
DEVICE "GSD device_19"  GSD.Device.PN
   slot 0: "Rack"  Rack  V1.0
   slot 0: "CPX_WP2_R"  CPX Rev 30  TN 197330  V4.2.30
      slot 0: "CPX Rev 30"  CPX Rev 30
      slot 1: "PN-IO Interface"  PN-IO Interface
         slot 1: "Port 1"  Port 1
         slot 2: "Port 2"  Port 2
   slot 1: "FB33 PNIO Module_1"  FB33 PNIO Module  TN 548755, CPX-FB33, Code F33
      slot 0: "FB33 PNIO Module"  FB33 PNIO Module
   slot 2: "MPA1S VMPA1-FB-EMS-8 [8DO]_1"  MPA1S VMPA1-FB-EMS-8 [8DO]  TN 533360, VMPA1-FB-EMS-8, Code A
      slot 0: "MPA1S VMPA1-FB-EMS-8 [8DO]"  MPA1S VMPA1-FB-EMS-8 [8DO]
   slot 3: "MPA1S VMPA1-FB-EMS-8 [8DO]_2"  MPA1S VMPA1-FB-EMS-8 [8DO]  TN 533360, VMPA1-FB-EMS-8, Code A
      slot 0: "MPA1S VMPA1-FB-EMS-8 [8DO]"  MPA1S VMPA1-FB-EMS-8 [8DO]
   slot 4: "MPA1S VMPA1-FB-EMS-8 [8DO]_3"  MPA1S VMPA1-FB-EMS-8 [8DO]  TN 533360, VMPA1-FB-EMS-8, Code A
      slot 0: "MPA1S VMPA1-FB-EMS-8 [8DO]"  MPA1S VMPA1-FB-EMS-8 [8DO]
   slot 5: "MPA1G VMPA1-FB-EMG-8 [8DO]_3"  MPA1G VMPA1-FB-EMG-8 [8DO]  TN 533361, VMPA1-FB-EMG-8, Code AH
      slot 0: "MPA1G VMPA1-FB-EMG-8 [8DO]"  MPA1G VMPA1-FB-EMG-8 [8DO]
DEVICE "GSD device_20"  GSD.Device.PN
   slot 0: "Rack"  Rack  V1.0
   slot 0: "CPX_TS_R"  CPX Rev 30  TN 197330  V4.2.30
      slot 0: "CPX Rev 30"  CPX Rev 30
      slot 1: "PN-IO Interface"  PN-IO Interface
         slot 1: "Port 1"  Port 1
         slot 2: "Port 2"  Port 2
   slot 1: "FB33 PNIO Module_1"  FB33 PNIO Module  TN 548755, CPX-FB33, Code F33
      slot 0: "FB33 PNIO Module"  FB33 PNIO Module
   slot 2: "MPA2S VMPA2-FB-EMS-4 [4DO]_1"  MPA2S VMPA2-FB-EMS-4 [4DO]  TN 537983, VMPA2-FB-EMS-4, Code B
      slot 0: "MPA2S VMPA2-FB-EMS-4 [4DO]"  MPA2S VMPA2-FB-EMS-4 [4DO]
   slot 3: "MPA2G VMPA2-FB-EMG-4 [4DO]_1"  MPA2G VMPA2-FB-EMG-4 [4DO]  TN 537984, VMPA2-FB-EMG-4, Code BH
      slot 0: "MPA2G VMPA2-FB-EMG-4 [4DO]"  MPA2G VMPA2-FB-EMG-4 [4DO]
   slot 4: "MPA1G VMPA1-FB-EMG-8 [8DO]_2"  MPA1G VMPA1-FB-EMG-8 [8DO]  TN 533361, VMPA1-FB-EMG-8, Code AH
      slot 0: "MPA1G VMPA1-FB-EMG-8 [8DO]"  MPA1G VMPA1-FB-EMG-8 [8DO]
   slot 5: "MPA1G VMPA1-FB-EMG-8 [8DO]_3"  MPA1G VMPA1-FB-EMG-8 [8DO]  TN 533361, VMPA1-FB-EMG-8, Code AH
      slot 0: "MPA1G VMPA1-FB-EMG-8 [8DO]"  MPA1G VMPA1-FB-EMG-8 [8DO]
   slot 6: "MPA1G VMPA1-FB-EMG-8 [8DO]_4"  MPA1G VMPA1-FB-EMG-8 [8DO]  TN 533361, VMPA1-FB-EMG-8, Code AH
      slot 0: "MPA1G VMPA1-FB-EMG-8 [8DO]"  MPA1G VMPA1-FB-EMG-8 [8DO]
   slot 7: "MPA1G VMPA1-FB-EMG-8 [8DO]_5"  MPA1G VMPA1-FB-EMG-8 [8DO]  TN 533361, VMPA1-FB-EMG-8, Code AH
      slot 0: "MPA1G VMPA1-FB-EMG-8 [8DO]"  MPA1G VMPA1-FB-EMG-8 [8DO]
   slot 8: "MPA1G VMPA1-FB-EMG-8 [8DO]_6"  MPA1G VMPA1-FB-EMG-8 [8DO]  TN 533361, VMPA1-FB-EMG-8, Code AH
      slot 0: "MPA1G VMPA1-FB-EMG-8 [8DO]"  MPA1G VMPA1-FB-EMG-8 [8DO]
DEVICE "GSD device_21"  GSD.Device.PN
   slot 0: "Rack"  Rack  V1.0
   slot 0: "CPX_WP5_R"  CPX Rev 30  TN 197330  V4.2.30
      slot 0: "CPX Rev 30"  CPX Rev 30
      slot 1: "PN-IO Interface"  PN-IO Interface
         slot 1: "Port 1"  Port 1
         slot 2: "Port 2"  Port 2
   slot 1: "FB33 PNIO Module_1"  FB33 PNIO Module  TN 548755, CPX-FB33, Code F33
      slot 0: "FB33 PNIO Module"  FB33 PNIO Module
   slot 2: "MPA1S VMPA1-FB-EMS-8 [8DO]_1"  MPA1S VMPA1-FB-EMS-8 [8DO]  TN 533360, VMPA1-FB-EMS-8, Code A
      slot 0: "MPA1S VMPA1-FB-EMS-8 [8DO]"  MPA1S VMPA1-FB-EMS-8 [8DO]
   slot 3: "MPA1S VMPA1-FB-EMS-8 [8DO]_2"  MPA1S VMPA1-FB-EMS-8 [8DO]  TN 533360, VMPA1-FB-EMS-8, Code A
      slot 0: "MPA1S VMPA1-FB-EMS-8 [8DO]"  MPA1S VMPA1-FB-EMS-8 [8DO]
   slot 4: "MPA1S VMPA1-FB-EMS-8 [8DO]_3"  MPA1S VMPA1-FB-EMS-8 [8DO]  TN 533360, VMPA1-FB-EMS-8, Code A
      slot 0: "MPA1S VMPA1-FB-EMS-8 [8DO]"  MPA1S VMPA1-FB-EMS-8 [8DO]
DEVICE "GSD device_22"  GSD.Device.PN
   slot 0: "Rack"  Rack  V1.0
   slot 0: "UR5_st4_R"  V1.0  00000
      slot 0: "V1.0"  V1.0
      slot 1: "Interface"  Interface
         slot 1: "RJ45 10/100 MBit/s"  RJ45 10/100 MBit/s
   slot 1: "1_T2O State"  1_T2O State  1.0
      slot 0: "1_T2O State"  1_T2O State
   slot 2: "2_T2O IO"  2_T2O IO  1.0
      slot 0: "2_T2O IO"  2_T2O IO
   slot 3: "3_T2O Joints"  3_T2O Joints  1.0
      slot 0: "3_T2O Joints"  3_T2O Joints
   slot 4: "4_T2O TCP"  4_T2O TCP  1.0
      slot 0: "4_T2O TCP"  4_T2O TCP
   slot 5: "5_T2O General Purpose Bit Registers"  5_T2O General Purpose Bit Registers  1.0
      slot 0: "5_T2O General Purpose Bit Registers"  5_T2O General Purpose Bit Registers
   slot 6: "6_T2O General Purpose Int Registers"  6_T2O General Purpose Int Registers  1.0
      slot 0: "6_T2O General Purpose Int Registers"  6_T2O General Purpose Int Registers
   slot 7: "7_T2O General Purpose Float Registers"  7_T2O General Purpose Float Registers  1.0
      slot 0: "7_T2O General Purpose Float Registers"  7_T2O General Purpose Float Registers
   slot 8: "8_O2T Robot IO"  8_O2T Robot IO  1.0
      slot 0: "8_O2T Robot IO"  8_O2T Robot IO
   slot 9: "9_O2T General Purpose Registers 1"  9_O2T General Purpose Registers 1  1.0
      slot 0: "9_O2T General Purpose Registers 1"  9_O2T General Purpose Registers 1
   slot 10: "10_O2T General Purpose Registers 2"  10_O2T General Purpose Registers 2  1.0
      slot 0: "10_O2T General Purpose Registers 2"  10_O2T General Purpose Registers 2
DEVICE "GSD device_15"  GSD.Device.PN
   slot 0: "Rack"  Rack  V1.0
   slot 0: "WP003-CAM-L"  In-Sight IS2XXX CC-B  IS2000-XXX  5.8.0
      slot 0: "In-Sight IS2XXX CC-B"  In-Sight IS2XXX CC-B  5.8.0
      slot 1: "Interface"  Interface
         slot 1: "Port 1"  Port 1
   slot 1: "Acquisition Control_1"  Acquisition Control  5.8.0
      slot 0: "Acquisition Control"  Acquisition Control  5.8.0
   slot 2: "Acquisition Status_1"  Acquisition Status  5.8.0
      slot 0: "Acquisition Status"  Acquisition Status  5.8.0
   slot 3: "Inspection Control_1"  Inspection Control  5.8.0
      slot 0: "Inspection Control"  Inspection Control  5.8.0
   slot 4: "Inspection Status_1"  Inspection Status  5.8.0
      slot 0: "Inspection Status"  Inspection Status  5.8.0
   slot 5: "Command Control_1"  Command Control  5.8.0
      slot 0: "Command Control"  Command Control  5.8.0
   slot 6: "SoftEvent Control_1"  SoftEvent Control  5.8.0
      slot 0: "SoftEvent Control"  SoftEvent Control  5.8.0
   slot 7: "User Data - 64 bytes_1"  User Data - 64 bytes  5.8.0
      slot 0: "User Data - 64 bytes"  User Data - 64 bytes  5.8.0
   slot 8: "Results - 64 bytes_1"  Results - 64 bytes  5.8.0
      slot 0: "Results - 64 bytes"  Results - 64 bytes  5.8.0
DEVICE "GSD device_3"  GSD.Device.PN
   slot 0: "Rack"  Rack  V1.0
   slot 0: "WP004-CAM-L"  In-Sight IS2XXX CC-B  IS2000-XXX  5.8.0
      slot 0: "In-Sight IS2XXX CC-B"  In-Sight IS2XXX CC-B  5.8.0
      slot 1: "Interface"  Interface
         slot 1: "Port 1"  Port 1
   slot 1: "Acquisition Control_1"  Acquisition Control  5.8.0
      slot 0: "Acquisition Control"  Acquisition Control  5.8.0
   slot 2: "Acquisition Status_1"  Acquisition Status  5.8.0
      slot 0: "Acquisition Status"  Acquisition Status  5.8.0
   slot 3: "Inspection Control_1"  Inspection Control  5.8.0
      slot 0: "Inspection Control"  Inspection Control  5.8.0
   slot 4: "Inspection Status_1"  Inspection Status  5.8.0
      slot 0: "Inspection Status"  Inspection Status  5.8.0
   slot 5: "Command Control_1"  Command Control  5.8.0
      slot 0: "Command Control"  Command Control  5.8.0
   slot 6: "SoftEvent Control_1"  SoftEvent Control  5.8.0
      slot 0: "SoftEvent Control"  SoftEvent Control  5.8.0
   slot 7: "User Data - 64 bytes_1"  User Data - 64 bytes  5.8.0
      slot 0: "User Data - 64 bytes"  User Data - 64 bytes  5.8.0
   slot 8: "Results - 64 bytes_1"  Results - 64 bytes  5.8.0
      slot 0: "Results - 64 bytes"  Results - 64 bytes  5.8.0
DEVICE "GSD device_23"  GSD.Device.PN
   slot 0: "Rack"  Rack  V1.0
   slot 0: "WP0031-DM8700-L"  DataMan 8700 CC-B  DMR-87xx-xx  6.2.0
      slot 0: "DataMan 8700 CC-B"  DataMan 8700 CC-B
      slot 1: "Interface"  Interface
         slot 1: "Port 1"  Port 1
   slot 1: "Acquisition Control_1"  Acquisition Control
      slot 0: "Acquisition Control"  Acquisition Control
   slot 2: "Acquisition Status_1"  Acquisition Status
      slot 0: "Acquisition Status"  Acquisition Status
   slot 3: "Results Control_1"  Results Control
      slot 0: "Results Control"  Results Control
   slot 4: "Results Status_1"  Results Status
      slot 0: "Results Status"  Results Status
   slot 5: "Soft Event Control_1"  Soft Event Control
      slot 0: "Soft Event Control"  Soft Event Control
   slot 6: "User Data - 64 bytes_1"  User Data - 64 bytes
      slot 0: "User Data - 64 bytes"  User Data - 64 bytes
   slot 7: "Result Data - 64 bytes_1"  Result Data - 64 bytes
      slot 0: "Result Data - 64 bytes"  Result Data - 64 bytes
DEVICE "GSD device_14"  GSD.Device.PN
   slot 0: "Rack"  Rack  V1.0
   slot 0: "WP002-DM8050-L"  DataMan 8000  DMR-8#00-0#00  5.4.2
      slot 0: "DataMan 8000"  DataMan 8000
      slot 1: "Interface"  Interface
         slot 1: "Port 1"  Port 1
   slot 1: "Acquisition Control_1"  Acquisition Control
      slot 0: "Acquisition Control"  Acquisition Control
   slot 2: "Acquisition Status_1"  Acquisition Status
      slot 0: "Acquisition Status"  Acquisition Status
   slot 3: "Results Control_1"  Results Control
      slot 0: "Results Control"  Results Control
   slot 4: "Results Status_1"  Results Status
      slot 0: "Results Status"  Results Status
   slot 5: "Soft Event Control_1"  Soft Event Control
      slot 0: "Soft Event Control"  Soft Event Control
   slot 6: "User Data - 64 bytes_1"  User Data - 64 bytes
      slot 0: "User Data - 64 bytes"  User Data - 64 bytes
   slot 7: "Result Data - 64 bytes_1"  Result Data - 64 bytes
      slot 0: "Result Data - 64 bytes"  Result Data - 64 bytes
DEVICE "GSD device_24"  GSD.Device.PN
   slot 0: "Rack"  Rack  V1.0
   slot 0: "WP002-DM8050-R"  DataMan 8000  DMR-8#00-0#00  5.4.2
      slot 0: "DataMan 8000"  DataMan 8000
      slot 1: "Interface"  Interface
         slot 1: "Port 1"  Port 1
   slot 1: "Acquisition Control_1"  Acquisition Control
      slot 0: "Acquisition Control"  Acquisition Control
   slot 2: "Acquisition Status_1"  Acquisition Status
      slot 0: "Acquisition Status"  Acquisition Status
   slot 3: "Results Control_1"  Results Control
      slot 0: "Results Control"  Results Control
   slot 4: "Results Status_1"  Results Status
      slot 0: "Results Status"  Results Status
   slot 5: "Soft Event Control_1"  Soft Event Control
      slot 0: "Soft Event Control"  Soft Event Control
   slot 6: "User Data - 64 bytes_1"  User Data - 64 bytes
      slot 0: "User Data - 64 bytes"  User Data - 64 bytes
   slot 7: "Result Data - 64 bytes_1"  Result Data - 64 bytes
      slot 0: "Result Data - 64 bytes"  Result Data - 64 bytes
DEVICE "GSD device_25"  GSD.Device.PN
   slot 0: "Rack"  Rack  V1.0
   slot 0: "WP001-DM8050-R"  DataMan 8000  DMR-8#00-0#00  5.4.2
      slot 0: "DataMan 8000"  DataMan 8000
      slot 1: "Interface"  Interface
         slot 1: "Port 1"  Port 1
   slot 1: "Acquisition Control_1"  Acquisition Control
      slot 0: "Acquisition Control"  Acquisition Control
   slot 2: "Acquisition Status_1"  Acquisition Status
      slot 0: "Acquisition Status"  Acquisition Status
   slot 3: "Results Control_1"  Results Control
      slot 0: "Results Control"  Results Control
   slot 4: "Results Status_1"  Results Status
      slot 0: "Results Status"  Results Status
   slot 5: "Soft Event Control_1"  Soft Event Control
      slot 0: "Soft Event Control"  Soft Event Control
   slot 6: "User Data - 64 bytes_1"  User Data - 64 bytes
      slot 0: "User Data - 64 bytes"  User Data - 64 bytes
   slot 7: "Result Data - 64 bytes_1"  Result Data - 64 bytes
      slot 0: "Result Data - 64 bytes"  Result Data - 64 bytes
DEVICE "GSD device_26"  GSD.Device.PN
   slot 0: "Rack"  Rack  V1.0
   slot 0: "WP001-DM260-R"  DataMan 260  DMR-260#-#0  5.5.0
      slot 0: "DataMan 260"  DataMan 260
      slot 1: "Interface"  Interface
         slot 1: "Port 1"  Port 1
   slot 1: "Acquisition Control_1"  Acquisition Control
      slot 0: "Acquisition Control"  Acquisition Control
   slot 2: "Acquisition Status_1"  Acquisition Status
      slot 0: "Acquisition Status"  Acquisition Status
   slot 3: "Results Control_1"  Results Control
      slot 0: "Results Control"  Results Control
   slot 4: "Results Status_1"  Results Status
      slot 0: "Results Status"  Results Status
   slot 5: "Soft Event Control_1"  Soft Event Control
      slot 0: "Soft Event Control"  Soft Event Control
   slot 6: "User Data - 64 bytes_1"  User Data - 64 bytes
      slot 0: "User Data - 64 bytes"  User Data - 64 bytes
   slot 7: "Result Data - 64 bytes_1"  Result Data - 64 bytes
      slot 0: "Result Data - 64 bytes"  Result Data - 64 bytes
DEVICE "GSD device_27"  GSD.Device.PN
   slot 0: "Rack"  Rack  V1.0
   slot 0: "WP002-DM260-r"  DataMan 260  DMR-260#-#0  5.5.0
      slot 0: "DataMan 260"  DataMan 260
      slot 1: "Interface"  Interface
         slot 1: "Port 1"  Port 1
   slot 1: "Acquisition Control_1"  Acquisition Control
      slot 0: "Acquisition Control"  Acquisition Control
   slot 2: "Acquisition Status_1"  Acquisition Status
      slot 0: "Acquisition Status"  Acquisition Status
   slot 3: "Results Control_1"  Results Control
      slot 0: "Results Control"  Results Control
   slot 4: "Results Status_1"  Results Status
      slot 0: "Results Status"  Results Status
   slot 5: "Soft Event Control_1"  Soft Event Control
      slot 0: "Soft Event Control"  Soft Event Control
   slot 6: "User Data - 64 bytes_1"  User Data - 64 bytes
      slot 0: "User Data - 64 bytes"  User Data - 64 bytes
   slot 7: "Result Data - 64 bytes_1"  Result Data - 64 bytes
      slot 0: "Result Data - 64 bytes"  Result Data - 64 bytes
DEVICE "GSD device_28"  GSD.Device.PN
   slot 0: "Rack"  Rack  V1.0
   slot 0: "WP003-DM260-r"  DataMan 260  DMR-260#-#0  5.5.0
      slot 0: "DataMan 260"  DataMan 260
      slot 1: "Interface"  Interface
         slot 1: "Port 1"  Port 1
   slot 1: "Acquisition Control_1"  Acquisition Control
      slot 0: "Acquisition Control"  Acquisition Control
   slot 2: "Acquisition Status_1"  Acquisition Status
      slot 0: "Acquisition Status"  Acquisition Status
   slot 3: "Results Control_1"  Results Control
      slot 0: "Results Control"  Results Control
   slot 4: "Results Status_1"  Results Status
      slot 0: "Results Status"  Results Status
   slot 5: "Soft Event Control_1"  Soft Event Control
      slot 0: "Soft Event Control"  Soft Event Control
   slot 6: "User Data - 64 bytes_1"  User Data - 64 bytes
      slot 0: "User Data - 64 bytes"  User Data - 64 bytes
   slot 7: "Result Data - 64 bytes_1"  Result Data - 64 bytes
      slot 0: "Result Data - 64 bytes"  Result Data - 64 bytes
DEVICE "GSD device_29"  GSD.Device.PN
   slot 0: "Rack"  Rack  V1.0
   slot 0: "WP0031-DM260-r"  DataMan 260  DMR-260#-#0  5.5.0
      slot 0: "DataMan 260"  DataMan 260
      slot 1: "Interface"  Interface
         slot 1: "Port 1"  Port 1
   slot 1: "Acquisition Control_1"  Acquisition Control
      slot 0: "Acquisition Control"  Acquisition Control
   slot 2: "Acquisition Status_1"  Acquisition Status
      slot 0: "Acquisition Status"  Acquisition Status
   slot 3: "Results Control_1"  Results Control
      slot 0: "Results Control"  Results Control
   slot 4: "Results Status_1"  Results Status
      slot 0: "Results Status"  Results Status
   slot 5: "Soft Event Control_1"  Soft Event Control
      slot 0: "Soft Event Control"  Soft Event Control
   slot 6: "User Data - 64 bytes_1"  User Data - 64 bytes
      slot 0: "User Data - 64 bytes"  User Data - 64 bytes
   slot 7: "Result Data - 64 bytes_1"  Result Data - 64 bytes
      slot 0: "Result Data - 64 bytes"  Result Data - 64 bytes
DEVICE "GSD device_30"  GSD.Device.PN
   slot 0: "Rack"  Rack  V1.0
   slot 0: "WP004-DM260-r"  DataMan 260  DMR-260#-#0  5.5.0
      slot 0: "DataMan 260"  DataMan 260
      slot 1: "Interface"  Interface
         slot 1: "Port 1"  Port 1
   slot 1: "Acquisition Control_1"  Acquisition Control
      slot 0: "Acquisition Control"  Acquisition Control
   slot 2: "Acquisition Status_1"  Acquisition Status
      slot 0: "Acquisition Status"  Acquisition Status
   slot 3: "Results Control_1"  Results Control
      slot 0: "Results Control"  Results Control
   slot 4: "Results Status_1"  Results Status
      slot 0: "Results Status"  Results Status
   slot 5: "Soft Event Control_1"  Soft Event Control
      slot 0: "Soft Event Control"  Soft Event Control
   slot 6: "User Data - 64 bytes_1"  User Data - 64 bytes
      slot 0: "User Data - 64 bytes"  User Data - 64 bytes
   slot 7: "Result Data - 64 bytes_1"  Result Data - 64 bytes
      slot 0: "Result Data - 64 bytes"  Result Data - 64 bytes
DEVICE "GSD device_31"  GSD.Device.PN
   slot 0: "Rack"  Rack  V1.0
   slot 0: "WP005-DM260-r"  DataMan 260  DMR-260#-#0  5.5.0
      slot 0: "DataMan 260"  DataMan 260
      slot 1: "Interface"  Interface
         slot 1: "Port 1"  Port 1
   slot 1: "Acquisition Control_1"  Acquisition Control
      slot 0: "Acquisition Control"  Acquisition Control
   slot 2: "Acquisition Status_1"  Acquisition Status
      slot 0: "Acquisition Status"  Acquisition Status
   slot 3: "Results Control_1"  Results Control
      slot 0: "Results Control"  Results Control
   slot 4: "Results Status_1"  Results Status
      slot 0: "Results Status"  Results Status
   slot 5: "Soft Event Control_1"  Soft Event Control
      slot 0: "Soft Event Control"  Soft Event Control
   slot 6: "User Data - 64 bytes_1"  User Data - 64 bytes
      slot 0: "User Data - 64 bytes"  User Data - 64 bytes
   slot 7: "Result Data - 64 bytes_1"  Result Data - 64 bytes
      slot 0: "Result Data - 64 bytes"  Result Data - 64 bytes
DEVICE "GSD device_32"  GSD.Device.PN
   slot 0: "Rack"  Rack  V1.0
   slot 0: "WP006-DM260-r"  DataMan 260  DMR-260#-#0  5.5.0
      slot 0: "DataMan 260"  DataMan 260
      slot 1: "Interface"  Interface
         slot 1: "Port 1"  Port 1
   slot 1: "Acquisition Control_1"  Acquisition Control
      slot 0: "Acquisition Control"  Acquisition Control
   slot 2: "Acquisition Status_1"  Acquisition Status
      slot 0: "Acquisition Status"  Acquisition Status
   slot 3: "Results Control_1"  Results Control
      slot 0: "Results Control"  Results Control
   slot 4: "Results Status_1"  Results Status
      slot 0: "Results Status"  Results Status
   slot 5: "Soft Event Control_1"  Soft Event Control
      slot 0: "Soft Event Control"  Soft Event Control
   slot 6: "User Data - 64 bytes_1"  User Data - 64 bytes
      slot 0: "User Data - 64 bytes"  User Data - 64 bytes
   slot 7: "Result Data - 64 bytes_1"  Result Data - 64 bytes
      slot 0: "Result Data - 64 bytes"  Result Data - 64 bytes
DEVICE "GSD device_33"  GSD.Device.PN
   slot 0: "Rack"  Rack  V1.0
   slot 0: "WP004-CAM-R"  In-Sight IS2XXX CC-B  IS2000-XXX  5.8.0
      slot 0: "In-Sight IS2XXX CC-B"  In-Sight IS2XXX CC-B  5.8.0
      slot 1: "Interface"  Interface
         slot 1: "Port 1"  Port 1
   slot 1: "Acquisition Control_1"  Acquisition Control  5.8.0
      slot 0: "Acquisition Control"  Acquisition Control  5.8.0
   slot 2: "Acquisition Status_1"  Acquisition Status  5.8.0
      slot 0: "Acquisition Status"  Acquisition Status  5.8.0
   slot 3: "Inspection Control_1"  Inspection Control  5.8.0
      slot 0: "Inspection Control"  Inspection Control  5.8.0
   slot 4: "Inspection Status_1"  Inspection Status  5.8.0
      slot 0: "Inspection Status"  Inspection Status  5.8.0
   slot 5: "Command Control_1"  Command Control  5.8.0
      slot 0: "Command Control"  Command Control  5.8.0
   slot 6: "SoftEvent Control_1"  SoftEvent Control  5.8.0
      slot 0: "SoftEvent Control"  SoftEvent Control  5.8.0
   slot 7: "User Data - 64 bytes_1"  User Data - 64 bytes  5.8.0
      slot 0: "User Data - 64 bytes"  User Data - 64 bytes  5.8.0
   slot 8: "Results - 64 bytes_1"  Results - 64 bytes  5.8.0
      slot 0: "Results - 64 bytes"  Results - 64 bytes  5.8.0
DEVICE "GSD device_34"  GSD.Device.PN
   slot 0: "Rack"  Rack  V1.0
   slot 0: "WP003-CAM-R"  In-Sight IS2XXX CC-B  IS2000-XXX  5.8.0
      slot 0: "In-Sight IS2XXX CC-B"  In-Sight IS2XXX CC-B  5.8.0
      slot 1: "Interface"  Interface
         slot 1: "Port 1"  Port 1
   slot 1: "Acquisition Control_1"  Acquisition Control  5.8.0
      slot 0: "Acquisition Control"  Acquisition Control  5.8.0
   slot 2: "Acquisition Status_1"  Acquisition Status  5.8.0
      slot 0: "Acquisition Status"  Acquisition Status  5.8.0
   slot 3: "Inspection Control_1"  Inspection Control  5.8.0
      slot 0: "Inspection Control"  Inspection Control  5.8.0
   slot 4: "Inspection Status_1"  Inspection Status  5.8.0
      slot 0: "Inspection Status"  Inspection Status  5.8.0
   slot 5: "Command Control_1"  Command Control  5.8.0
      slot 0: "Command Control"  Command Control  5.8.0
   slot 6: "SoftEvent Control_1"  SoftEvent Control  5.8.0
      slot 0: "SoftEvent Control"  SoftEvent Control  5.8.0
   slot 7: "User Data - 64 bytes_1"  User Data - 64 bytes  5.8.0
      slot 0: "User Data - 64 bytes"  User Data - 64 bytes  5.8.0
   slot 8: "Results - 64 bytes_1"  Results - 64 bytes  5.8.0
      slot 0: "Results - 64 bytes"  Results - 64 bytes  5.8.0
DEVICE "GSD device_35"  GSD.Device.PN
   slot 0: "Rack"  Rack  V1.0
   slot 0: "WP0031-DM8700-r"  DataMan 8700 CC-B  DMR-87xx-xx  6.2.0
      slot 0: "DataMan 8700 CC-B"  DataMan 8700 CC-B
      slot 1: "Interface"  Interface
         slot 1: "Port 1"  Port 1
   slot 1: "Acquisition Control_1"  Acquisition Control
      slot 0: "Acquisition Control"  Acquisition Control
   slot 2: "Acquisition Status_1"  Acquisition Status
      slot 0: "Acquisition Status"  Acquisition Status
   slot 3: "Results Control_1"  Results Control
      slot 0: "Results Control"  Results Control
   slot 4: "Results Status_1"  Results Status
      slot 0: "Results Status"  Results Status
   slot 5: "Soft Event Control_1"  Soft Event Control
      slot 0: "Soft Event Control"  Soft Event Control
   slot 6: "User Data - 64 bytes_1"  User Data - 64 bytes
      slot 0: "User Data - 64 bytes"  User Data - 64 bytes
   slot 7: "Result Data - 64 bytes_1"  Result Data - 64 bytes
      slot 0: "Result Data - 64 bytes"  Result Data - 64 bytes
DEVICE "GSD device_36"  GSD.Device.PN
   slot 0: "Rack"  Rack  V1.0
   slot 0: "WP004-DM8050-r"  DataMan 8000  DMR-8#00-0#00  5.4.2
      slot 0: "DataMan 8000"  DataMan 8000
      slot 1: "Interface"  Interface
         slot 1: "Port 1"  Port 1
   slot 1: "Acquisition Control_1"  Acquisition Control
      slot 0: "Acquisition Control"  Acquisition Control
   slot 2: "Acquisition Status_1"  Acquisition Status
      slot 0: "Acquisition Status"  Acquisition Status
   slot 3: "Results Control_1"  Results Control
      slot 0: "Results Control"  Results Control
   slot 4: "Results Status_1"  Results Status
      slot 0: "Results Status"  Results Status
   slot 5: "Soft Event Control_1"  Soft Event Control
      slot 0: "Soft Event Control"  Soft Event Control
   slot 6: "User Data - 64 bytes_1"  User Data - 64 bytes
      slot 0: "User Data - 64 bytes"  User Data - 64 bytes
   slot 7: "Result Data - 64 bytes_1"  Result Data - 64 bytes
      slot 0: "Result Data - 64 bytes"  Result Data - 64 bytes
DEVICE "GSD device_37"  GSD.Device.PN
   slot 0: "Rack"  Rack  V1.0
   slot 0: "CPX_Rack_L"  CPX Rev 30  TN 197330  V4.2.30
      slot 0: "CPX Rev 30"  CPX Rev 30
      slot 1: "PN-IO Interface"  PN-IO Interface
         slot 1: "Port 1"  Port 1
         slot 2: "Port 2"  Port 2
   slot 1: "FB33 PNIO Module_1"  FB33 PNIO Module  TN 548755, CPX-FB33, Code F33
      slot 0: "FB33 PNIO Module"  FB33 PNIO Module
   slot 2: "16DI [16DI]_1"  16DI [16DI]  TN 543815, CPX-16DI, Code M
      slot 0: "16DI [16DI]"  16DI [16DI]
   slot 3: "16DI [16DI]_2"  16DI [16DI]  TN 543815, CPX-16DI, Code M
      slot 0: "16DI [16DI]"  16DI [16DI]
   slot 4: "16DI [16DI]_3"  16DI [16DI]  TN 543815, CPX-16DI, Code M
      slot 0: "16DI [16DI]"  16DI [16DI]
   slot 5: "16DI [16DI]_4"  16DI [16DI]  TN 543815, CPX-16DI, Code M
      slot 0: "16DI [16DI]"  16DI [16DI]
   slot 6: "16DI [16DI]_5"  16DI [16DI]  TN 543815, CPX-16DI, Code M
      slot 0: "16DI [16DI]"  16DI [16DI]
   slot 7: "MPA1S VMPA1-FB-EMS-8 [8DO]_1"  MPA1S VMPA1-FB-EMS-8 [8DO]  TN 533360, VMPA1-FB-EMS-8, Code A
      slot 0: "MPA1S VMPA1-FB-EMS-8 [8DO]"  MPA1S VMPA1-FB-EMS-8 [8DO]
   slot 8: "MPA1S VMPA1-FB-EMS-8 [8DO]_2"  MPA1S VMPA1-FB-EMS-8 [8DO]  TN 533360, VMPA1-FB-EMS-8, Code A
      slot 0: "MPA1S VMPA1-FB-EMS-8 [8DO]"  MPA1S VMPA1-FB-EMS-8 [8DO]
   slot 9: "MPA1S VMPA1-FB-EMS-8 [8DO]_3"  MPA1S VMPA1-FB-EMS-8 [8DO]  TN 533360, VMPA1-FB-EMS-8, Code A
      slot 0: "MPA1S VMPA1-FB-EMS-8 [8DO]"  MPA1S VMPA1-FB-EMS-8 [8DO]
   slot 10: "MPA1S VMPA1-FB-EMS-8 [8DO]_4"  MPA1S VMPA1-FB-EMS-8 [8DO]  TN 533360, VMPA1-FB-EMS-8, Code A
      slot 0: "MPA1S VMPA1-FB-EMS-8 [8DO]"  MPA1S VMPA1-FB-EMS-8 [8DO]
   slot 11: "MPA1S VMPA1-FB-EMS-8 [8DO]_5"  MPA1S VMPA1-FB-EMS-8 [8DO]  TN 533360, VMPA1-FB-EMS-8, Code A
      slot 0: "MPA1S VMPA1-FB-EMS-8 [8DO]"  MPA1S VMPA1-FB-EMS-8 [8DO]
DEVICE "GSD device_38"  GSD.Device.PN
   slot 0: "Rack"  Rack  V1.0
   slot 0: "CPX_Rack_R"  CPX Rev 30  TN 197330  V4.2.30
      slot 0: "CPX Rev 30"  CPX Rev 30
      slot 1: "PN-IO Interface"  PN-IO Interface
         slot 1: "Port 1"  Port 1
         slot 2: "Port 2"  Port 2
   slot 1: "FB33 PNIO Module_1"  FB33 PNIO Module  TN 548755, CPX-FB33, Code F33
      slot 0: "FB33 PNIO Module"  FB33 PNIO Module
   slot 2: "16DI [16DI]_1"  16DI [16DI]  TN 543815, CPX-16DI, Code M
      slot 0: "16DI [16DI]"  16DI [16DI]
   slot 3: "16DI [16DI]_2"  16DI [16DI]  TN 543815, CPX-16DI, Code M
      slot 0: "16DI [16DI]"  16DI [16DI]
   slot 4: "16DI [16DI]_3"  16DI [16DI]  TN 543815, CPX-16DI, Code M
      slot 0: "16DI [16DI]"  16DI [16DI]
   slot 5: "16DI [16DI]_4"  16DI [16DI]  TN 543815, CPX-16DI, Code M
      slot 0: "16DI [16DI]"  16DI [16DI]
   slot 6: "16DI [16DI]_5"  16DI [16DI]  TN 543815, CPX-16DI, Code M
      slot 0: "16DI [16DI]"  16DI [16DI]
   slot 7: "MPA1S VMPA1-FB-EMS-8 [8DO]_1"  MPA1S VMPA1-FB-EMS-8 [8DO]  TN 533360, VMPA1-FB-EMS-8, Code A
      slot 0: "MPA1S VMPA1-FB-EMS-8 [8DO]"  MPA1S VMPA1-FB-EMS-8 [8DO]
   slot 8: "MPA1S VMPA1-FB-EMS-8 [8DO]_2"  MPA1S VMPA1-FB-EMS-8 [8DO]  TN 533360, VMPA1-FB-EMS-8, Code A
      slot 0: "MPA1S VMPA1-FB-EMS-8 [8DO]"  MPA1S VMPA1-FB-EMS-8 [8DO]
   slot 9: "MPA1S VMPA1-FB-EMS-8 [8DO]_4"  MPA1S VMPA1-FB-EMS-8 [8DO]  TN 533360, VMPA1-FB-EMS-8, Code A
      slot 0: "MPA1S VMPA1-FB-EMS-8 [8DO]"  MPA1S VMPA1-FB-EMS-8 [8DO]
   slot 10: "MPA1S VMPA1-FB-EMS-8 [8DO]_3"  MPA1S VMPA1-FB-EMS-8 [8DO]  TN 533360, VMPA1-FB-EMS-8, Code A
      slot 0: "MPA1S VMPA1-FB-EMS-8 [8DO]"  MPA1S VMPA1-FB-EMS-8 [8DO]
   slot 11: "MPA1S VMPA1-FB-EMS-8 [8DO]_5"  MPA1S VMPA1-FB-EMS-8 [8DO]  TN 533360, VMPA1-FB-EMS-8, Code A
      slot 0: "MPA1S VMPA1-FB-EMS-8 [8DO]"  MPA1S VMPA1-FB-EMS-8 [8DO]
DEVICE "GSD device_39"  GSD.Device.PN
   slot 0: "Rack"  Rack  V1.0
   slot 0: "WP000-DM260-L"  DataMan 260  DMR-260#-#0  5.5.0
      slot 0: "DataMan 260"  DataMan 260
      slot 1: "Interface"  Interface
         slot 1: "Port 1"  Port 1
   slot 1: "Acquisition Control_1"  Acquisition Control
      slot 0: "Acquisition Control"  Acquisition Control
   slot 2: "Acquisition Status_1"  Acquisition Status
      slot 0: "Acquisition Status"  Acquisition Status
   slot 3: "Results Control_1"  Results Control
      slot 0: "Results Control"  Results Control
   slot 4: "Results Status_1"  Results Status
      slot 0: "Results Status"  Results Status
   slot 5: "Soft Event Control_1"  Soft Event Control
      slot 0: "Soft Event Control"  Soft Event Control
   slot 6: "User Data - 64 bytes_1"  User Data - 64 bytes
      slot 0: "User Data - 64 bytes"  User Data - 64 bytes
   slot 7: "Result Data - 64 bytes_1"  Result Data - 64 bytes
      slot 0: "Result Data - 64 bytes"  Result Data - 64 bytes
DEVICE "GSD device_40"  GSD.Device.PN
   slot 0: "Rack"  Rack  V1.0
   slot 0: "WP000-DM8050-L"  DataMan 8000  DMR-8#00-0#00  5.4.2
      slot 0: "DataMan 8000"  DataMan 8000
      slot 1: "Interface"  Interface
         slot 1: "Port 1"  Port 1
   slot 1: "Acquisition Control_1"  Acquisition Control
      slot 0: "Acquisition Control"  Acquisition Control
   slot 2: "Acquisition Status_1"  Acquisition Status
      slot 0: "Acquisition Status"  Acquisition Status
   slot 3: "Results Control_1"  Results Control
      slot 0: "Results Control"  Results Control
   slot 4: "Results Status_1"  Results Status
      slot 0: "Results Status"  Results Status
   slot 5: "Soft Event Control_1"  Soft Event Control
      slot 0: "Soft Event Control"  Soft Event Control
   slot 6: "User Data - 64 bytes_1"  User Data - 64 bytes
      slot 0: "User Data - 64 bytes"  User Data - 64 bytes
   slot 7: "Result Data - 64 bytes_1"  Result Data - 64 bytes
      slot 0: "Result Data - 64 bytes"  Result Data - 64 bytes
DEVICE "GSD device_41"  GSD.Device.PN
   slot 0: "Rack"  Rack  V1.0
   slot 0: "WP000-DM260-R"  DataMan 260  DMR-260#-#0  5.5.0
      slot 0: "DataMan 260"  DataMan 260
      slot 1: "Interface"  Interface
         slot 1: "Port 1"  Port 1
   slot 1: "Acquisition Control_1"  Acquisition Control
      slot 0: "Acquisition Control"  Acquisition Control
   slot 2: "Acquisition Status_1"  Acquisition Status
      slot 0: "Acquisition Status"  Acquisition Status
   slot 3: "Results Control_1"  Results Control
      slot 0: "Results Control"  Results Control
   slot 4: "Results Status_1"  Results Status
      slot 0: "Results Status"  Results Status
   slot 5: "Soft Event Control_1"  Soft Event Control
      slot 0: "Soft Event Control"  Soft Event Control
   slot 6: "User Data - 64 bytes_1"  User Data - 64 bytes
      slot 0: "User Data - 64 bytes"  User Data - 64 bytes
   slot 7: "Result Data - 64 bytes_1"  Result Data - 64 bytes
      slot 0: "Result Data - 64 bytes"  Result Data - 64 bytes
DEVICE "GSD device_42"  GSD.Device.PN
   slot 0: "Rack"  Rack  V1.0
   slot 0: "WP000-DM8050-R"  DataMan 8000  DMR-8#00-0#00  5.4.2
      slot 0: "DataMan 8000"  DataMan 8000
      slot 1: "Interface"  Interface
         slot 1: "Port 1"  Port 1
   slot 1: "Acquisition Control_1"  Acquisition Control
      slot 0: "Acquisition Control"  Acquisition Control
   slot 2: "Acquisition Status_1"  Acquisition Status
      slot 0: "Acquisition Status"  Acquisition Status
   slot 3: "Results Control_1"  Results Control
      slot 0: "Results Control"  Results Control
   slot 4: "Results Status_1"  Results Status
      slot 0: "Results Status"  Results Status
   slot 5: "Soft Event Control_1"  Soft Event Control
      slot 0: "Soft Event Control"  Soft Event Control
   slot 6: "User Data - 64 bytes_1"  User Data - 64 bytes
      slot 0: "User Data - 64 bytes"  User Data - 64 bytes
   slot 7: "Result Data - 64 bytes_1"  Result Data - 64 bytes
      slot 0: "Result Data - 64 bytes"  Result Data - 64 bytes
DEVICE "S71500/ET200MP station_2"  S7-1500 station
   slot 0: "Rail_0"  Rack  6ES7 590-1***0-0AA0
   slot 1: "PLC_LINE_L"  CPU 1517-3 PN/DP  6ES7 517-3AP00-0AB0  V2.8
      slot 3: "CPU display_1"  6ES7591-1BA00-0AA0
      slot 32768: "PROFINET interface_1"  X1
         slot 32769: "Port_1"  X1 P1
         slot 32770: "Port_2"  X1 P2
      slot 33024: "PROFINET interface_2"  X2
         slot 33025: "Port_1"  X2 P1
      slot 33280: "DP interface_1"  X3
      slot 34817: "Virtual CP interface port_1"  Virtual CP interface port  Virtual CP interface port
DEVICE "S71500/ET200MP station_1"  S7-1500 station
   slot 0: "Rail_0"  Rack  6ES7 590-1***0-0AA0
   slot 1: "PLC_LINE_R"  CPU 1517-3 PN/DP  6ES7 517-3AP00-0AB0  V2.8
      slot 3: "CPU display_1"  6ES7591-1BA00-0AA0
      slot 32768: "PROFINET interface_1"  X1
         slot 32769: "Port_1"  X1 P1
         slot 32770: "Port_2"  X1 P2
      slot 33024: "PROFINET interface_2"  X2
         slot 33025: "Port_1"  X2 P1
      slot 33280: "DP interface_1"  X3
      slot 34817: "Virtual CP interface port_1"  Virtual CP interface port  Virtual CP interface port
*)

// ===== PLC "PLC_LINE_L"  CPU 1517-3 PN/DP =====

VAR_GLOBAL   // PLC tag table "Default tag table"
   "Clock_Byte" AT %MB0 : Byte;
   "Clock_10Hz" AT %M0.0 : Bool;
   "Clock_5Hz" AT %M0.1 : Bool;
   "Clock_2.5Hz" AT %M0.2 : Bool;
   "Clock_2Hz" AT %M0.3 : Bool;
   "Clock_1.25Hz" AT %M0.4 : Bool;
   "Clock_1Hz" AT %M0.5 : Bool;
   "Clock_0.625Hz" AT %M0.6 : Bool;
   "Clock_0.5Hz" AT %M0.7 : Bool;
   "System_Byte" AT %MB1 : Byte;
   "FirstScan" AT %M1.0 : Bool;
   "DiagStatusUpdate" AT %M1.1 : Bool;
   "AlwaysTRUE" AT %M1.2 : Bool;
   "AlwaysFALSE" AT %M1.3 : Bool;
END_VAR

ORGANIZATION_BLOCK "Main"   // OB1, LAD, ProgramCycle
TITLE = "Main Program Sweep (Cycle)"
{ S7_Optimized_Access := 'TRUE' }
VERSION : 0.1
   VAR_INPUT
      Initial_Call : Bool;   // Initial call of this OB
      Remanence : Bool;   // =True, if remanent data are available
   END_VAR
BEGIN
END_ORGANIZATION_BLOCK

// ===== PLC "PLC_LINE_R"  CPU 1517-3 PN/DP =====

VAR_GLOBAL   // PLC tag table "Default tag table"
   "Clock_Byte" AT %MB0 : Byte;
   "Clock_10Hz" AT %M0.0 : Bool;
   "Clock_5Hz" AT %M0.1 : Bool;
   "Clock_2.5Hz" AT %M0.2 : Bool;
   "Clock_2Hz" AT %M0.3 : Bool;
   "Clock_1.25Hz" AT %M0.4 : Bool;
   "Clock_1Hz" AT %M0.5 : Bool;
   "Clock_0.625Hz" AT %M0.6 : Bool;
   "Clock_0.5Hz" AT %M0.7 : Bool;
   "System_Byte" AT %MB1 : Byte;
   "FirstScan" AT %M1.0 : Bool;
   "DiagStatusUpdate" AT %M1.1 : Bool;
   "AlwaysTRUE" AT %M1.2 : Bool;
   "AlwaysFALSE" AT %M1.3 : Bool;
END_VAR

ORGANIZATION_BLOCK "Main"   // OB1, LAD, ProgramCycle
TITLE = "Main Program Sweep (Cycle)"
{ S7_Optimized_Access := 'TRUE' }
VERSION : 0.1
   VAR_INPUT
      Initial_Call : Bool;   // Initial call of this OB
      Remanence : Bool;   // =True, if remanent data are available
   END_VAR
BEGIN
END_ORGANIZATION_BLOCK